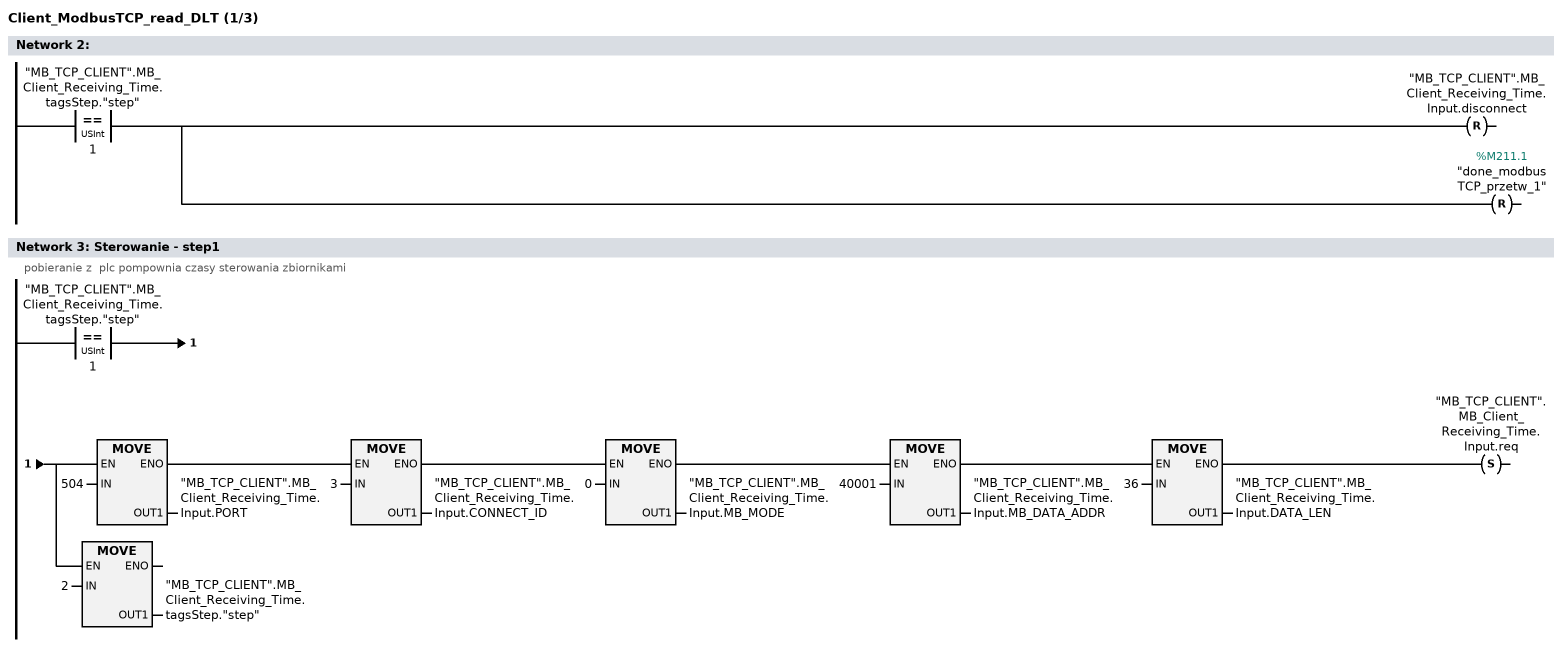
   RUNG wire#powerrail
      { S7_Templates := "SrcType := USInt" } EQ_Contact(in1 := "MB_TCP_CLIENT".MB_Client_Receiving_Time.tagsStep."step", in2 := 1)
      wire#w1
      R_Coil( "MB_TCP_CLIENT".MB_Client_Receiving_Time.Input.disconnect )
   END_RUNG
   RUNG wire#w1
      R_Coil( "done_modbusTCP_przetw_1" )
   END_RUNG
   // the same network as SCL:
   IF "MB_TCP_CLIENT".MB_Client_Receiving_Time.tagsStep."step" = 1 THEN
       "MB_TCP_CLIENT".MB_Client_Receiving_Time.Input.disconnect := FALSE;
       "done_modbusTCP_przetw_1" := FALSE;
   END_IF;
END_REGION

REGION Network 3: Sterowanie - step1
   // pobieranie z  plc pompownia czasy sterowania zbiornikami
   RUNG wire#powerrail
      { S7_Templates := "SrcType := USInt" } EQ_Contact(in1 := "MB_TCP_CLIENT".MB_Client_Receiving_Time.tagsStep."step", in2 := 1)
      wire#w1
      { S7_GenerateENO := "TRUE" } Move(in := 504, out1 => "MB_TCP_CLIENT".MB_Client_Receiving_Time.Input.PORT)
      { S7_GenerateENO := "TRUE" } Move(in := 3, out1 => "MB_TCP_CLIENT".MB_Client_Receiving_Time.Input.CONNECT_ID)
      { S7_GenerateENO := "TRUE" } Move(in := 0, out1 => "MB_TCP_CLIENT".MB_Client_Receiving_Time.Input.MB_MODE)
      { S7_GenerateENO := "TRUE" } Move(in := 40001, out1 => "MB_TCP_CLIENT".MB_Client_Receiving_Time.Input.MB_DATA_ADDR)
      { S7_GenerateENO := "TRUE" } Move(in := 36, out1 => "MB_TCP_CLIENT".MB_Client_Receiving_Time.Input.DATA_LEN)
      S_Coil( "MB_TCP_CLIENT".MB_Client_Receiving_Time.Input.req )
   END_RUNG
   RUNG wire#w1
      { S7_GenerateENO := "TRUE" } Move(in := 2, out1 => "MB_TCP_CLIENT".MB_Client_Receiving_Time.tagsStep."step")
   END_RUNG
   // the same network as SCL:
   // ENO of a box is taken as its EN; it also drops when the box reports an error
   IF "MB_TCP_CLIENT".MB_Client_Receiving_Time.tagsStep."step" = 1 THEN
       "MB_TCP_CLIENT".MB_Client_Receiving_Time.Input.PORT := 504;
       "MB_TCP_CLIENT".MB_Client_Receiving_Time.Input.CONNECT_ID := 3;
       "MB_TCP_CLIENT".MB_Client_Receiving_Time.Input.MB_MODE := 0;
       "MB_TCP_CLIENT".MB_Client_Receiving_Time.Input.MB_DATA_ADDR := 40001;
       "MB_TCP_CLIENT".MB_Client_Receiving_Time.Input.DATA_LEN := 36;
       "MB_TCP_CLIENT".MB_Client_Receiving_Time.Input.req := TRUE;
       "MB_TCP_CLIENT".MB_Client_Receiving_Time.tagsStep."step" := 2;
   END_IF;
END_REGION

REGION Network 4: step 2
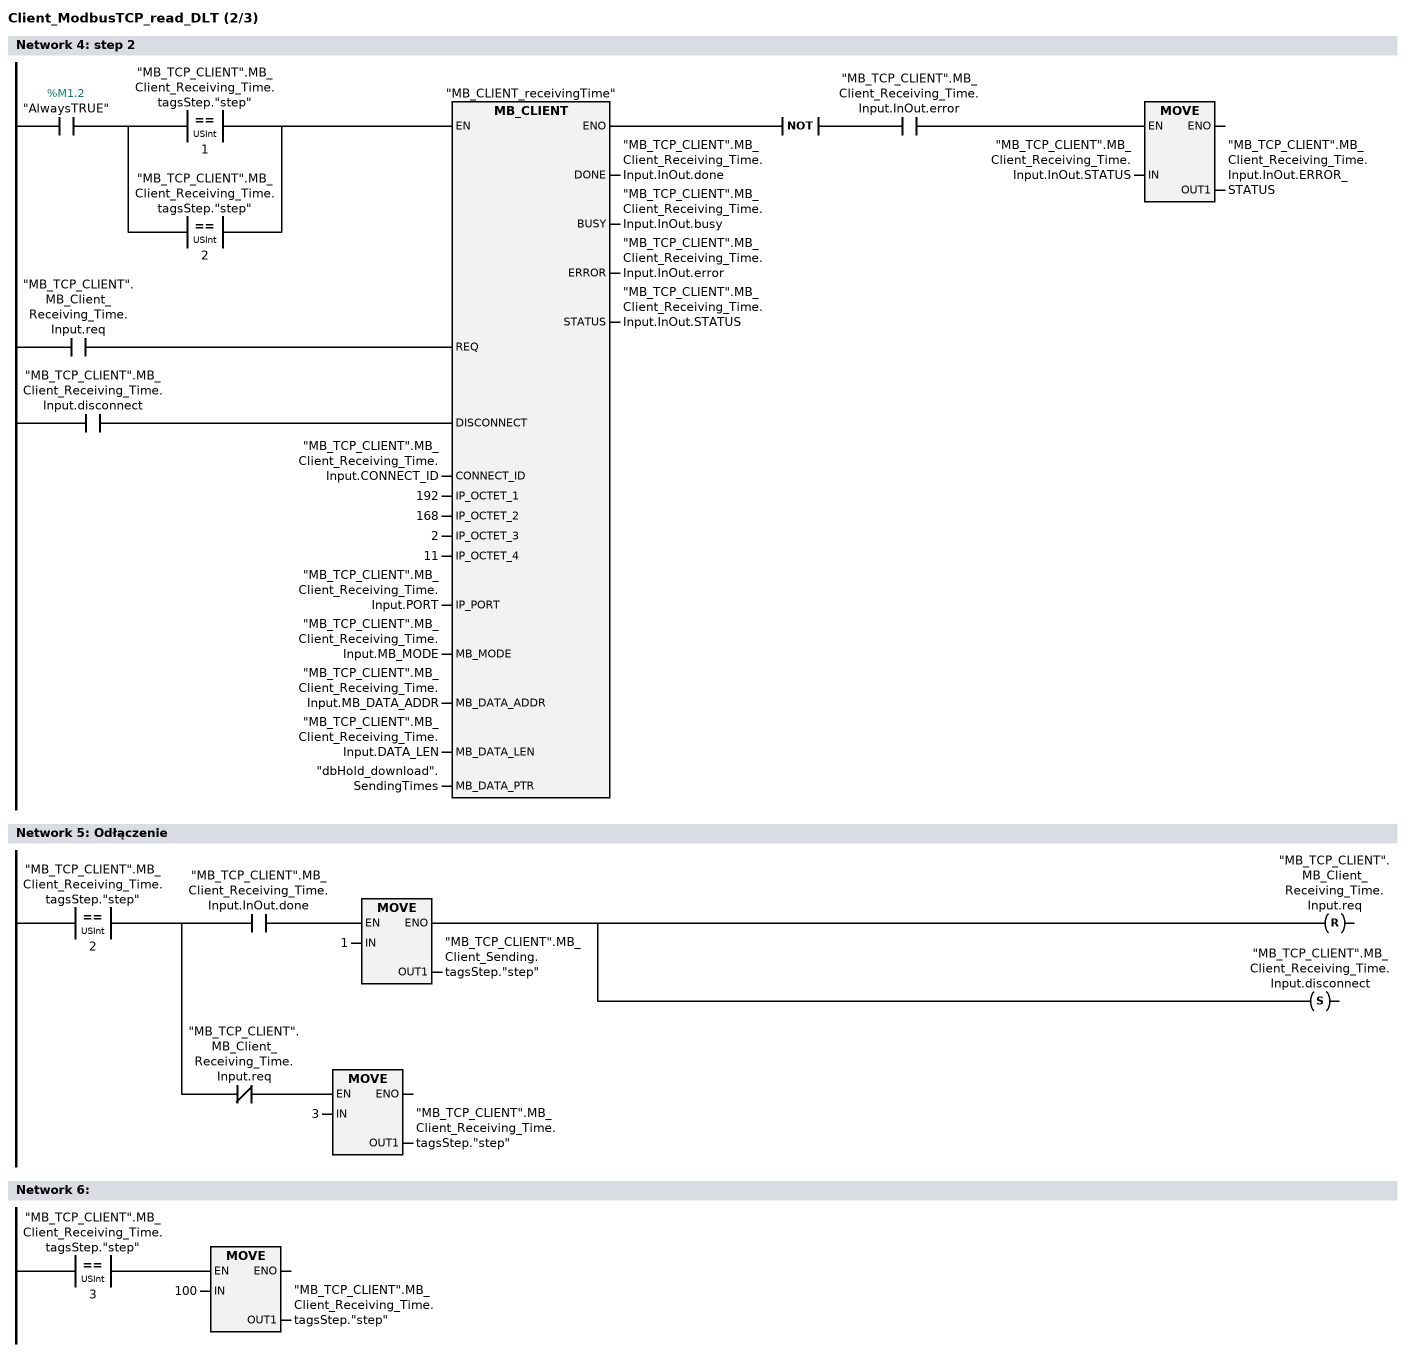
   RUNG wire#powerrail
      Contact( "AlwaysTRUE" )
      wire#w1
      { S7_Templates := "SrcType := USInt" } EQ_Contact(in1 := "MB_TCP_CLIENT".MB_Client_Receiving_Time.tagsStep."step", in2 := 1)
      wire#w2
      { S7_Templates := "[card1200 := 1, card1500 := 0]" } "MB_CLIENT_receivingTime".MB_CLIENT(REQ := wire#w3, DISCONNECT := wire#w4, CONNECT_ID := "MB_TCP_CLIENT".MB_Client_Receiving_Time.Input.CONNECT_ID, IP_OCTET_1 := 192, IP_OCTET_2 := 168, IP_OCTET_3 := 2, IP_OCTET_4 := 11, IP_PORT := "MB_TCP_CLIENT".MB_Client_Receiving_Time.Input.PORT, MB_MODE := "MB_TCP_CLIENT".MB_Client_Receiving_Time.Input.MB_MODE, MB_DATA_ADDR := "MB_TCP_CLIENT".MB_Client_Receiving_Time.Input.MB_DATA_ADDR, MB_DATA_LEN := "MB_TCP_CLIENT".MB_Client_Receiving_Time.Input.DATA_LEN, MB_DATA_PTR := "dbHold_download".SendingTimes, DONE => "MB_TCP_CLIENT".MB_Client_Receiving_Time.Input.InOut.done, BUSY => "MB_TCP_CLIENT".MB_Client_Receiving_Time.Input.InOut.busy, ERROR => "MB_TCP_CLIENT".MB_Client_Receiving_Time.Input.InOut.error, STATUS => "MB_TCP_CLIENT".MB_Client_Receiving_Time.Input.InOut.STATUS)
      Not()
      Contact( "MB_TCP_CLIENT".MB_Client_Receiving_Time.Input.InOut.error )
      Move(in := "MB_TCP_CLIENT".MB_Client_Receiving_Time.Input.InOut.STATUS, out1 => "MB_TCP_CLIENT".MB_Client_Receiving_Time.Input.InOut.ERROR_STATUS)
   END_RUNG
   RUNG wire#w1
      { S7_Templates := "SrcType := USInt" } EQ_Contact(in1 := "MB_TCP_CLIENT".MB_Client_Receiving_Time.tagsStep."step", in2 := 2)
   END_RUNG wire#w2
   RUNG wire#powerrail
      Contact( "MB_TCP_CLIENT".MB_Client_Receiving_Time.Input.req )
   END_RUNG wire#w3
   RUNG wire#powerrail
      Contact( "MB_TCP_CLIENT".MB_Client_Receiving_Time.Input.disconnect )
   END_RUNG wire#w4
   // the same network as SCL:
   #_w1 := "AlwaysTRUE" AND (("MB_TCP_CLIENT".MB_Client_Receiving_Time.tagsStep."step" = 1) OR ("MB_TCP_CLIENT".MB_Client_Receiving_Time.tagsStep."step" = 2));
   "MB_CLIENT_receivingTime"(EN := #_w1,   // MB_CLIENT
                           REQ := "MB_TCP_CLIENT".MB_Client_Receiving_Time.Input.req,
                           DISCONNECT := "MB_TCP_CLIENT".MB_Client_Receiving_Time.Input.disconnect,
                           CONNECT_ID := "MB_TCP_CLIENT".MB_Client_Receiving_Time.Input.CONNECT_ID,
                           IP_OCTET_1 := 192,
                           IP_OCTET_2 := 168,
                           IP_OCTET_3 := 2,
                           IP_OCTET_4 := 11,
                           IP_PORT := "MB_TCP_CLIENT".MB_Client_Receiving_Time.Input.PORT,
                           MB_MODE := "MB_TCP_CLIENT".MB_Client_Receiving_Time.Input.MB_MODE,
                           MB_DATA_ADDR := "MB_TCP_CLIENT".MB_Client_Receiving_Time.Input.MB_DATA_ADDR,
                           MB_DATA_LEN := "MB_TCP_CLIENT".MB_Client_Receiving_Time.Input.DATA_LEN,
                           MB_DATA_PTR := "dbHold_download".SendingTimes,
                           DONE => "MB_TCP_CLIENT".MB_Client_Receiving_Time.Input.InOut.done,
                           BUSY => "MB_TCP_CLIENT".MB_Client_Receiving_Time.Input.InOut.busy,
                           ERROR => "MB_TCP_CLIENT".MB_Client_Receiving_Time.Input.InOut.error,
                           STATUS => "MB_TCP_CLIENT".MB_Client_Receiving_Time.Input.InOut.STATUS,
                           ENO => #_w2);
   IF NOT #_w2 AND "MB_TCP_CLIENT".MB_Client_Receiving_Time.Input.InOut.error THEN
       "MB_TCP_CLIENT".MB_Client_Receiving_Time.Input.InOut.ERROR_STATUS := "MB_TCP_CLIENT".MB_Client_Receiving_Time.Input.InOut.STATUS;
   END_IF;
END_REGION

REGION Network 5: Odłączenie
   RUNG wire#powerrail
      { S7_Templates := "SrcType := USInt" } EQ_Contact(in1 := "MB_TCP_CLIENT".MB_Client_Receiving_Time.tagsStep."step", in2 := 2)
      wire#w1
      Contact( "MB_TCP_CLIENT".MB_Client_Receiving_Time.Input.InOut.done )
      Move(in := 1, out1 => "MB_TCP_CLIENT".MB_Client_Sending.tagsStep."step")
      wire#w2
      R_Coil( "MB_TCP_CLIENT".MB_Client_Receiving_Time.Input.req )
   END_RUNG
   RUNG wire#w2
      S_Coil( "MB_TCP_CLIENT".MB_Client_Receiving_Time.Input.disconnect )
   END_RUNG
   RUNG wire#w1
      I_Contact( "MB_TCP_CLIENT".MB_Client_Receiving_Time.Input.req )
      Move(in := 3, out1 => "MB_TCP_CLIENT".MB_Client_Receiving_Time.tagsStep."step")
   END_RUNG
   // the same network as SCL:
   #_w1 := "MB_TCP_CLIENT".MB_Client_Receiving_Time.tagsStep."step" = 2;
   IF #_w1 AND "MB_TCP_CLIENT".MB_Client_Receiving_Time.Input.InOut.done THEN
       "MB_TCP_CLIENT".MB_Client_Sending.tagsStep."step" := 1;
       "MB_TCP_CLIENT".MB_Client_Receiving_Time.Input.req := FALSE;
       "MB_TCP_CLIENT".MB_Client_Receiving_Time.Input.disconnect := TRUE;
   END_IF;
   IF #_w1 AND NOT "MB_TCP_CLIENT".MB_Client_Receiving_Time.Input.req THEN
       "MB_TCP_CLIENT".MB_Client_Receiving_Time.tagsStep."step" := 3;
   END_IF;
END_REGION

REGION Network 6
   RUNG wire#powerrail
      { S7_Templates := "SrcType := USInt" } EQ_Contact(in1 := "MB_TCP_CLIENT".MB_Client_Receiving_Time.tagsStep."step", in2 := 3)
      Move(in := 100, out1 => "MB_TCP_CLIENT".MB_Client_Receiving_Time.tagsStep."step")
   END_RUNG
   // the same network as SCL:
   IF "MB_TCP_CLIENT".MB_Client_Receiving_Time.tagsStep."step" = 3 THEN
       "MB_TCP_CLIENT".MB_Client_Receiving_Time.tagsStep."step" := 100;
   END_IF;
END_REGION

REGION Network 7
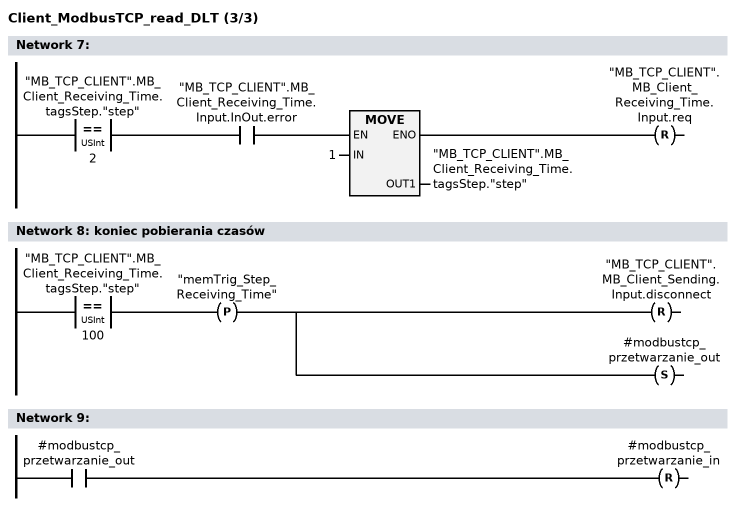
   RUNG wire#powerrail
      { S7_Templates := "SrcType := USInt" } EQ_Contact(in1 := "MB_TCP_CLIENT".MB_Client_Receiving_Time.tagsStep."step", in2 := 2)
      Contact( "MB_TCP_CLIENT".MB_Client_Receiving_Time.Input.InOut.error )
      Move(in := 1, out1 => "MB_TCP_CLIENT".MB_Client_Receiving_Time.tagsStep."step")
      R_Coil( "MB_TCP_CLIENT".MB_Client_Receiving_Time.Input.req )
   END_RUNG
   // the same network as SCL:
   #_w1 := ("MB_TCP_CLIENT".MB_Client_Receiving_Time.tagsStep."step" = 2) AND "MB_TCP_CLIENT".MB_Client_Receiving_Time.Input.InOut.error;
   IF #_w1 THEN
       "MB_TCP_CLIENT".MB_Client_Receiving_Time.tagsStep."step" := 1;
       "MB_TCP_CLIENT".MB_Client_Receiving_Time.Input.req := FALSE;
   END_IF;
END_REGION

REGION Network 8: koniec pobierania czasów
   RUNG wire#powerrail
      { S7_Templates := "SrcType := USInt" } EQ_Contact(in1 := "MB_TCP_CLIENT".MB_Client_Receiving_Time.tagsStep."step", in2 := 100)
      P_Trig( "memTrig_Step_Receiving_Time" )
      wire#w1
      R_Coil( "MB_TCP_CLIENT".MB_Client_Sending.Input.disconnect )
   END_RUNG
   RUNG wire#w1
      S_Coil( #modbustcp_przetwarzanie_out )
   END_RUNG
   // the same network as SCL:
   #_w1 := "MB_TCP_CLIENT".MB_Client_Receiving_Time.tagsStep."step" = 100;
   #_w2 := #_w1 AND NOT "memTrig_Step_Receiving_Time";   // rising edge
   "memTrig_Step_Receiving_Time" := #_w1;
   IF #_w2 THEN
       "MB_TCP_CLIENT".MB_Client_Sending.Input.disconnect := FALSE;
       #modbustcp_przetwarzanie_out := TRUE;
   END_IF;
END_REGION

REGION Network 9
   RUNG wire#powerrail
      Contact( #modbustcp_przetwarzanie_out )
      R_Coil( #modbustcp_przetwarzanie_in )
   END_RUNG
   // the same network as SCL:
   IF #modbustcp_przetwarzanie_out THEN #modbustcp_przetwarzanie_in := FALSE; END_IF;
END_REGION
END_FUNCTION_BLOCK

FUNCTION_BLOCK "Client_ModbusTCP_sending_analogs"   // FB4, LAD
TITLE = Wysyłanie analogów
{ S7_Optimized_Access := 'TRUE' }
AUTHOR : rtecmer
VERSION : 0.1
// Wysyłanie pomiarów
// stored: AutoNumber true, IsIECCheckEnabled false, IsRetainMemResEnabled false, MemoryReserve 250, SetENOAutomatically false, UDAEnableTagReadback false
   VAR_IN_OUT
      modbustcp_przetwarzanie_in : Bool;
      modbustcp_przetwarzanie_out : Bool;
   END_VAR
   VAR_TEMP   // added for the SCL form of the ladder/FBD networks
      _w1 : Bool;
      _w2 : Bool;
   END_VAR
BEGIN

REGION Network 2: Inicjacja modbus po błędzie i restarcie
END_REGION

REGION Network 3
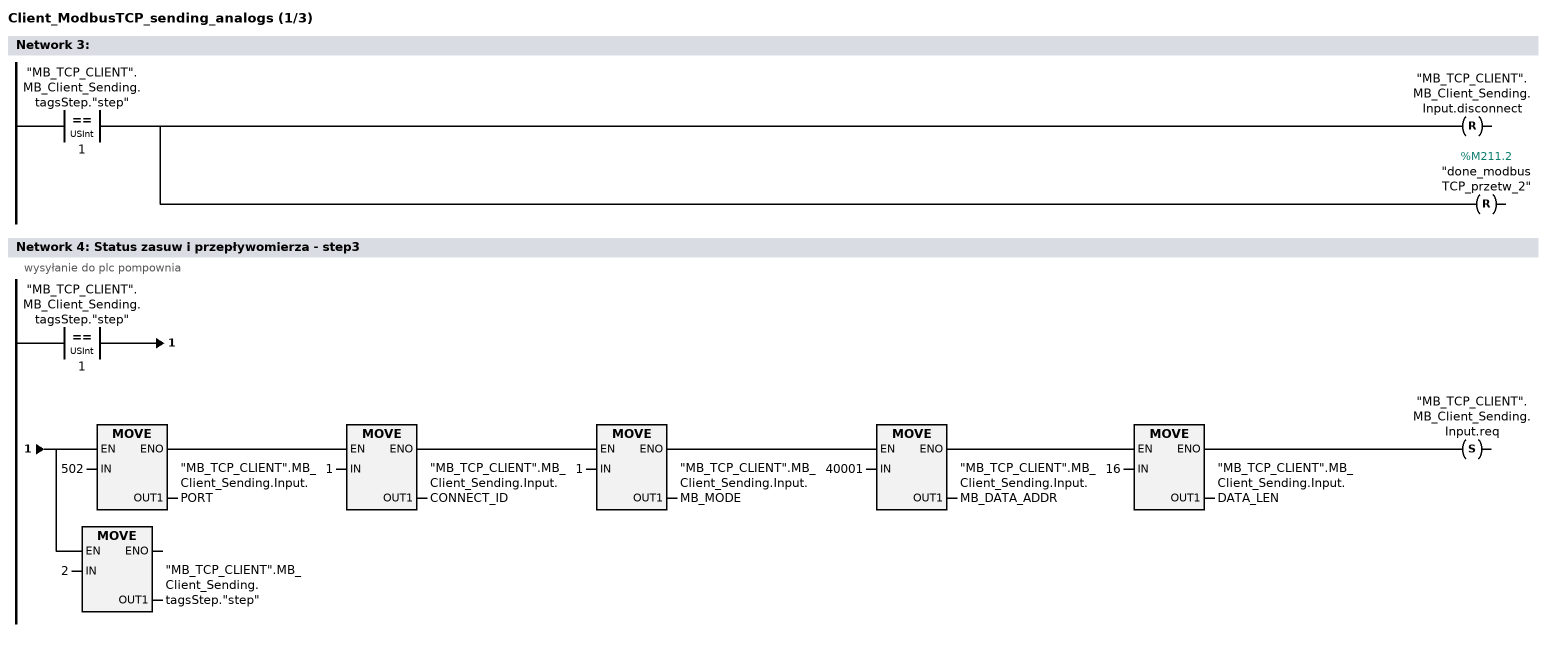
   RUNG wire#powerrail
      { S7_Templates := "SrcType := USInt" } EQ_Contact(in1 := "MB_TCP_CLIENT".MB_Client_Sending.tagsStep."step", in2 := 1)
      wire#w1
      R_Coil( "MB_TCP_CLIENT".MB_Client_Sending.Input.disconnect )
   END_RUNG
   RUNG wire#w1
      R_Coil( "done_modbusTCP_przetw_2" )
   END_RUNG
   // the same network as SCL:
   IF "MB_TCP_CLIENT".MB_Client_Sending.tagsStep."step" = 1 THEN
       "MB_TCP_CLIENT".MB_Client_Sending.Input.disconnect := FALSE;
       "done_modbusTCP_przetw_2" := FALSE;
   END_IF;
END_REGION

REGION Network 4: Status zasuw i przepływomierza - step3
   // wysyłanie do plc pompownia
   RUNG wire#powerrail
      { S7_Templates := "SrcType := USInt" } EQ_Contact(in1 := "MB_TCP_CLIENT".MB_Client_Sending.tagsStep."step", in2 := 1)
      wire#w1
      { S7_GenerateENO := "TRUE" } Move(in := 502, out1 => "MB_TCP_CLIENT".MB_Client_Sending.Input.PORT)
      { S7_GenerateENO := "TRUE" } Move(in := 1, out1 => "MB_TCP_CLIENT".MB_Client_Sending.Input.CONNECT_ID)
      { S7_GenerateENO := "TRUE" } Move(in := 1, out1 => "MB_TCP_CLIENT".MB_Client_Sending.Input.MB_MODE)
      { S7_GenerateENO := "TRUE" } Move(in := 40001, out1 => "MB_TCP_CLIENT".MB_Client_Sending.Input.MB_DATA_ADDR)
      { S7_GenerateENO := "TRUE" } Move(in := 16, out1 => "MB_TCP_CLIENT".MB_Client_Sending.Input.DATA_LEN)
      S_Coil( "MB_TCP_CLIENT".MB_Client_Sending.Input.req )
   END_RUNG
   RUNG wire#w1
      { S7_GenerateENO := "TRUE" } Move(in := 2, out1 => "MB_TCP_CLIENT".MB_Client_Sending.tagsStep."step")
   END_RUNG
   // the same network as SCL:
   // ENO of a box is taken as its EN; it also drops when the box reports an error
   IF "MB_TCP_CLIENT".MB_Client_Sending.tagsStep."step" = 1 THEN
       "MB_TCP_CLIENT".MB_Client_Sending.Input.PORT := 502;
       "MB_TCP_CLIENT".MB_Client_Sending.Input.CONNECT_ID := 1;
       "MB_TCP_CLIENT".MB_Client_Sending.Input.MB_MODE := 1;
       "MB_TCP_CLIENT".MB_Client_Sending.Input.MB_DATA_ADDR := 40001;
       "MB_TCP_CLIENT".MB_Client_Sending.Input.DATA_LEN := 16;
       "MB_TCP_CLIENT".MB_Client_Sending.Input.req := TRUE;
       "MB_TCP_CLIENT".MB_Client_Sending.tagsStep."step" := 2;
   END_IF;
END_REGION

REGION Network 5: step 3
   // Analogi
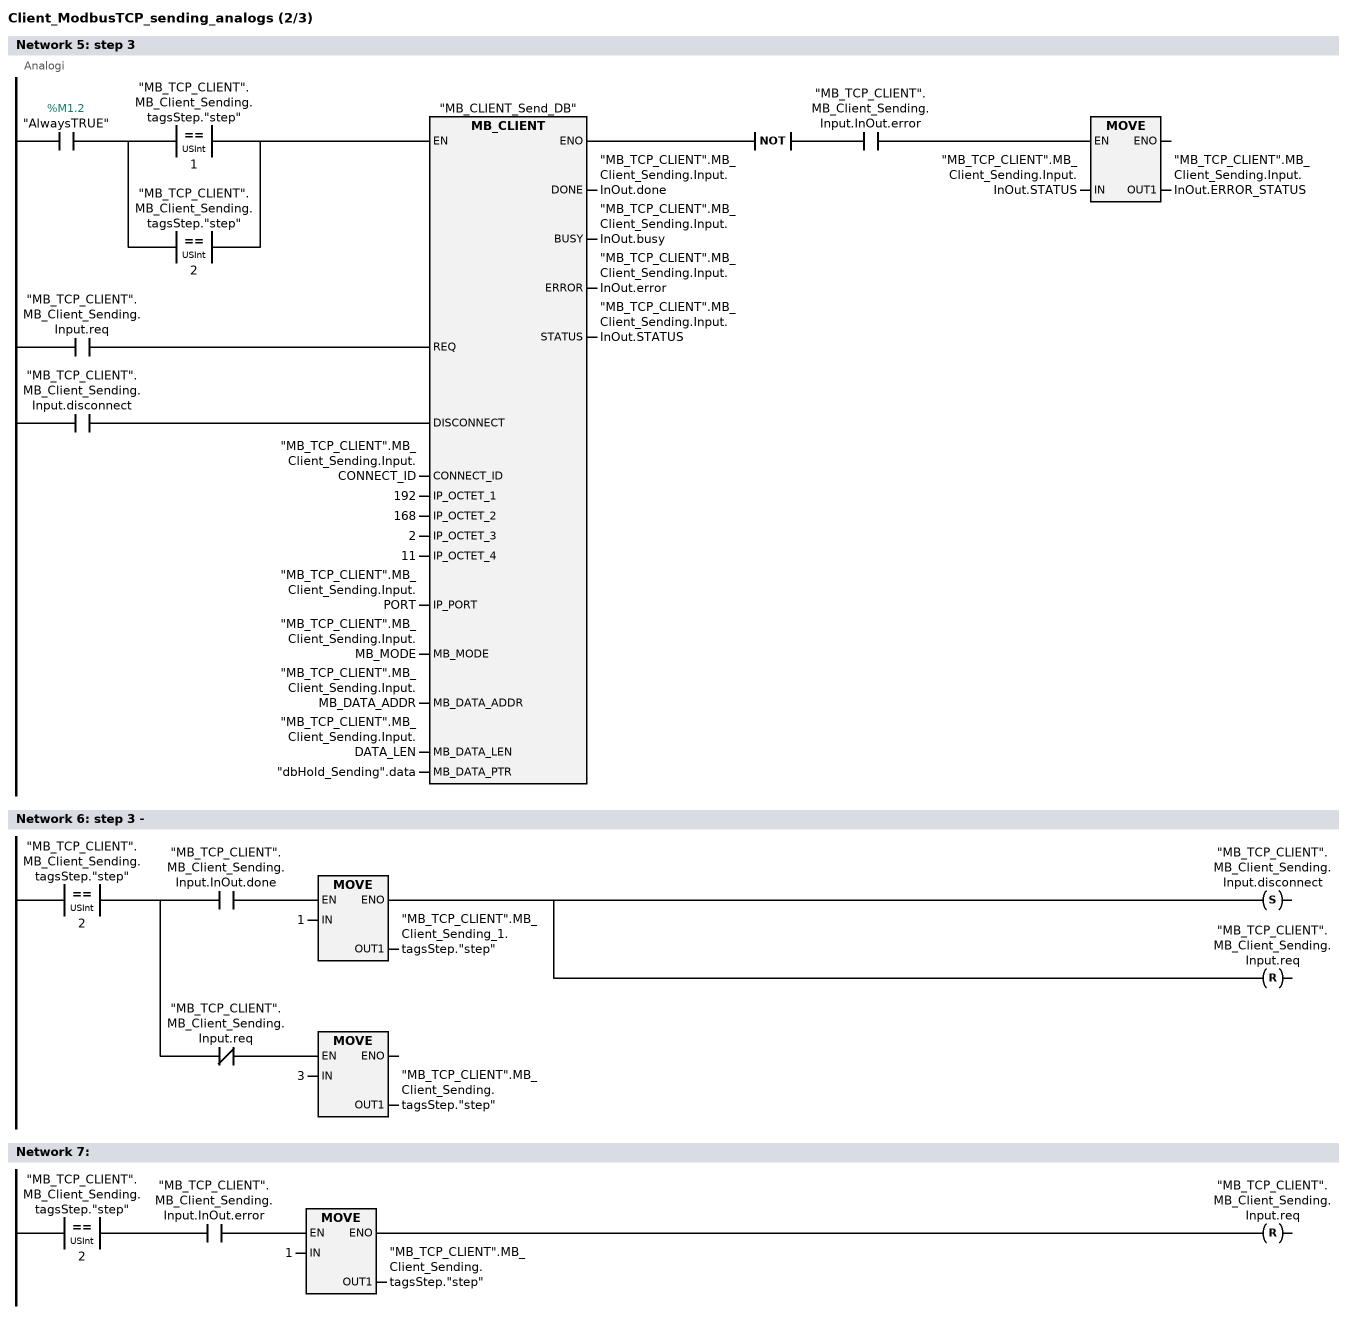
   RUNG wire#powerrail
      Contact( "AlwaysTRUE" )
      wire#w1
      { S7_Templates := "SrcType := USInt" } EQ_Contact(in1 := "MB_TCP_CLIENT".MB_Client_Sending.tagsStep."step", in2 := 1)
      wire#w2
      { S7_Templates := "[card1200 := 1, card1500 := 0]" } "MB_CLIENT_Send_DB".MB_CLIENT(REQ := wire#w3, DISCONNECT := wire#w4, CONNECT_ID := "MB_TCP_CLIENT".MB_Client_Sending.Input.CONNECT_ID, IP_OCTET_1 := 192, IP_OCTET_2 := 168, IP_OCTET_3 := 2, IP_OCTET_4 := 11, IP_PORT := "MB_TCP_CLIENT".MB_Client_Sending.Input.PORT, MB_MODE := "MB_TCP_CLIENT".MB_Client_Sending.Input.MB_MODE, MB_DATA_ADDR := "MB_TCP_CLIENT".MB_Client_Sending.Input.MB_DATA_ADDR, MB_DATA_LEN := "MB_TCP_CLIENT".MB_Client_Sending.Input.DATA_LEN, MB_DATA_PTR := "dbHold_Sending".data, DONE => "MB_TCP_CLIENT".MB_Client_Sending.Input.InOut.done, BUSY => "MB_TCP_CLIENT".MB_Client_Sending.Input.InOut.busy, ERROR => "MB_TCP_CLIENT".MB_Client_Sending.Input.InOut.error, STATUS => "MB_TCP_CLIENT".MB_Client_Sending.Input.InOut.STATUS)
      Not()
      Contact( "MB_TCP_CLIENT".MB_Client_Sending.Input.InOut.error )
      Move(in := "MB_TCP_CLIENT".MB_Client_Sending.Input.InOut.STATUS, out1 => "MB_TCP_CLIENT".MB_Client_Sending.Input.InOut.ERROR_STATUS)
   END_RUNG
   RUNG wire#w1
      { S7_Templates := "SrcType := USInt" } EQ_Contact(in1 := "MB_TCP_CLIENT".MB_Client_Sending.tagsStep."step", in2 := 2)
   END_RUNG wire#w2
   RUNG wire#powerrail
      Contact( "MB_TCP_CLIENT".MB_Client_Sending.Input.req )
   END_RUNG wire#w3
   RUNG wire#powerrail
      Contact( "MB_TCP_CLIENT".MB_Client_Sending.Input.disconnect )
   END_RUNG wire#w4
   // the same network as SCL:
   #_w1 := "AlwaysTRUE" AND (("MB_TCP_CLIENT".MB_Client_Sending.tagsStep."step" = 1) OR ("MB_TCP_CLIENT".MB_Client_Sending.tagsStep."step" = 2));
   "MB_CLIENT_Send_DB"(EN := #_w1,   // MB_CLIENT
                       REQ := "MB_TCP_CLIENT".MB_Client_Sending.Input.req,
                       DISCONNECT := "MB_TCP_CLIENT".MB_Client_Sending.Input.disconnect,
                       CONNECT_ID := "MB_TCP_CLIENT".MB_Client_Sending.Input.CONNECT_ID,
                       IP_OCTET_1 := 192,
                       IP_OCTET_2 := 168,
                       IP_OCTET_3 := 2,
                       IP_OCTET_4 := 11,
                       IP_PORT := "MB_TCP_CLIENT".MB_Client_Sending.Input.PORT,
                       MB_MODE := "MB_TCP_CLIENT".MB_Client_Sending.Input.MB_MODE,
                       MB_DATA_ADDR := "MB_TCP_CLIENT".MB_Client_Sending.Input.MB_DATA_ADDR,
                       MB_DATA_LEN := "MB_TCP_CLIENT".MB_Client_Sending.Input.DATA_LEN,
                       MB_DATA_PTR := "dbHold_Sending".data,
                       DONE => "MB_TCP_CLIENT".MB_Client_Sending.Input.InOut.done,
                       BUSY => "MB_TCP_CLIENT".MB_Client_Sending.Input.InOut.busy,
                       ERROR => "MB_TCP_CLIENT".MB_Client_Sending.Input.InOut.error,
                       STATUS => "MB_TCP_CLIENT".MB_Client_Sending.Input.InOut.STATUS,
                       ENO => #_w2);
   IF NOT #_w2 AND "MB_TCP_CLIENT".MB_Client_Sending.Input.InOut.error THEN
       "MB_TCP_CLIENT".MB_Client_Sending.Input.InOut.ERROR_STATUS := "MB_TCP_CLIENT".MB_Client_Sending.Input.InOut.STATUS;
   END_IF;
END_REGION

REGION Network 6: step 3 -
   RUNG wire#powerrail
      { S7_Templates := "SrcType := USInt" } EQ_Contact(in1 := "MB_TCP_CLIENT".MB_Client_Sending.tagsStep."step", in2 := 2)
      wire#w1
      Contact( "MB_TCP_CLIENT".MB_Client_Sending.Input.InOut.done )
      Move(in := 1, out1 => "MB_TCP_CLIENT".MB_Client_Sending_1.tagsStep."step")
      wire#w2
      S_Coil( "MB_TCP_CLIENT".MB_Client_Sending.Input.disconnect )
   END_RUNG
   RUNG wire#w2
      R_Coil( "MB_TCP_CLIENT".MB_Client_Sending.Input.req )
   END_RUNG
   RUNG wire#w1
      I_Contact( "MB_TCP_CLIENT".MB_Client_Sending.Input.req )
      Move(in := 3, out1 => "MB_TCP_CLIENT".MB_Client_Sending.tagsStep."step")
   END_RUNG
   // the same network as SCL:
   #_w1 := "MB_TCP_CLIENT".MB_Client_Sending.tagsStep."step" = 2;
   IF #_w1 AND "MB_TCP_CLIENT".MB_Client_Sending.Input.InOut.done THEN
       "MB_TCP_CLIENT".MB_Client_Sending_1.tagsStep."step" := 1;
       "MB_TCP_CLIENT".MB_Client_Sending.Input.disconnect := TRUE;
       "MB_TCP_CLIENT".MB_Client_Sending.Input.req := FALSE;
   END_IF;
   IF #_w1 AND NOT "MB_TCP_CLIENT".MB_Client_Sending.Input.req THEN
       "MB_TCP_CLIENT".MB_Client_Sending.tagsStep."step" := 3;
   END_IF;
END_REGION

REGION Network 7
   RUNG wire#powerrail
      { S7_Templates := "SrcType := USInt" } EQ_Contact(in1 := "MB_TCP_CLIENT".MB_Client_Sending.tagsStep."step", in2 := 2)
      Contact( "MB_TCP_CLIENT".MB_Client_Sending.Input.InOut.error )
      Move(in := 1, out1 => "MB_TCP_CLIENT".MB_Client_Sending.tagsStep."step")
      R_Coil( "MB_TCP_CLIENT".MB_Client_Sending.Input.req )
   END_RUNG
   // the same network as SCL:
   #_w1 := ("MB_TCP_CLIENT".MB_Client_Sending.tagsStep."step" = 2) AND "MB_TCP_CLIENT".MB_Client_Sending.Input.InOut.error;
   IF #_w1 THEN
       "MB_TCP_CLIENT".MB_Client_Sending.tagsStep."step" := 1;
       "MB_TCP_CLIENT".MB_Client_Sending.Input.req := FALSE;
   END_IF;
END_REGION

REGION Network 8
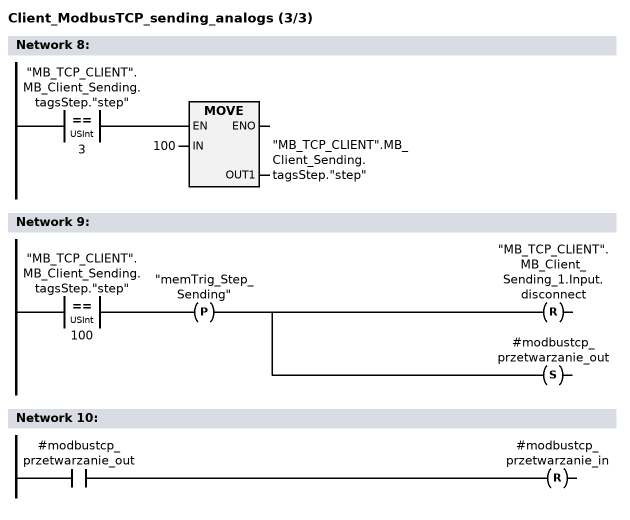
   RUNG wire#powerrail
      { S7_Templates := "SrcType := USInt" } EQ_Contact(in1 := "MB_TCP_CLIENT".MB_Client_Sending.tagsStep."step", in2 := 3)
      Move(in := 100, out1 => "MB_TCP_CLIENT".MB_Client_Sending.tagsStep."step")
   END_RUNG
   // the same network as SCL:
   IF "MB_TCP_CLIENT".MB_Client_Sending.tagsStep."step" = 3 THEN
       "MB_TCP_CLIENT".MB_Client_Sending.tagsStep."step" := 100;
   END_IF;
END_REGION

REGION Network 9
   RUNG wire#powerrail
      { S7_Templates := "SrcType := USInt" } EQ_Contact(in1 := "MB_TCP_CLIENT".MB_Client_Sending.tagsStep."step", in2 := 100)
      P_Trig( "memTrig_Step_Sending" )
      wire#w1
      R_Coil( "MB_TCP_CLIENT".MB_Client_Sending_1.Input.disconnect )
   END_RUNG
   RUNG wire#w1
      S_Coil( #modbustcp_przetwarzanie_out )
   END_RUNG
   // the same network as SCL:
   #_w1 := "MB_TCP_CLIENT".MB_Client_Sending.tagsStep."step" = 100;
   #_w2 := #_w1 AND NOT "memTrig_Step_Sending";   // rising edge
   "memTrig_Step_Sending" := #_w1;
   IF #_w2 THEN
       "MB_TCP_CLIENT".MB_Client_Sending_1.Input.disconnect := FALSE;
       #modbustcp_przetwarzanie_out := TRUE;
   END_IF;
END_REGION

REGION Network 10
   RUNG wire#powerrail
      Contact( #modbustcp_przetwarzanie_out )
      R_Coil( #modbustcp_przetwarzanie_in )
   END_RUNG
   // the same network as SCL:
   IF #modbustcp_przetwarzanie_out THEN #modbustcp_przetwarzanie_in := FALSE; END_IF;
END_REGION
END_FUNCTION_BLOCK

FUNCTION_BLOCK "Client_ModbusTCP_sending_status"   // FB8, LAD
TITLE = Przekazanie statusu utrządzeń
{ S7_Optimized_Access := 'TRUE' }
AUTHOR : rtecmer
VERSION : 0.1
// funkcja przesyła na server status urządzeńz PLC 2 Zbiorniki
// stored: AutoNumber true, IsIECCheckEnabled false, IsRetainMemResEnabled false, MemoryReserve 250, SetENOAutomatically false, UDAEnableTagReadback false
   VAR_IN_OUT
      modbustcp_przetwarzanie_in : Bool;
      modbustcp_przetwarzanie_out : Bool;
   END_VAR
   VAR_TEMP   // added for the SCL form of the ladder/FBD networks
      _w1 : Bool;
      _w2 : Bool;
   END_VAR
BEGIN

REGION Network 1: Inicjacja modbus po błędzie i restarcie
END_REGION

REGION Network 2
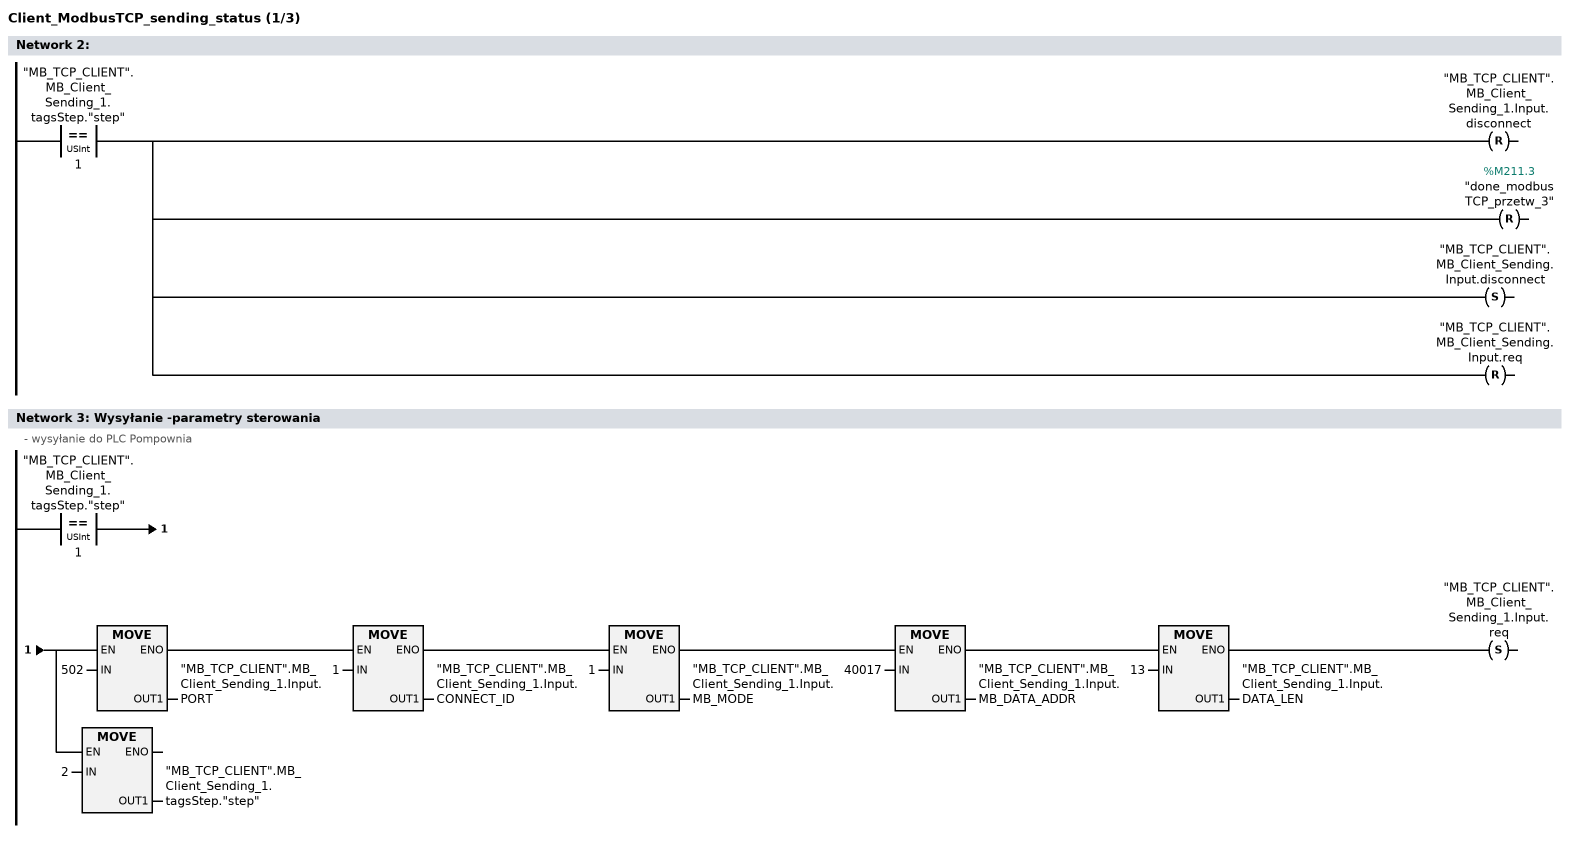
   RUNG wire#powerrail
      { S7_Templates := "SrcType := USInt" } EQ_Contact(in1 := "MB_TCP_CLIENT".MB_Client_Sending_1.tagsStep."step", in2 := 1)
      wire#w1
      R_Coil( "MB_TCP_CLIENT".MB_Client_Sending_1.Input.disconnect )
   END_RUNG
   RUNG wire#w1
      R_Coil( "done_modbusTCP_przetw_3" )
   END_RUNG
   RUNG wire#w1
      S_Coil( "MB_TCP_CLIENT".MB_Client_Sending.Input.disconnect )
   END_RUNG
   RUNG wire#w1
      R_Coil( "MB_TCP_CLIENT".MB_Client_Sending.Input.req )
   END_RUNG
   // the same network as SCL:
   IF "MB_TCP_CLIENT".MB_Client_Sending_1.tagsStep."step" = 1 THEN
       "MB_TCP_CLIENT".MB_Client_Sending_1.Input.disconnect := FALSE;
       "done_modbusTCP_przetw_3" := FALSE;
       "MB_TCP_CLIENT".MB_Client_Sending.Input.disconnect := TRUE;
       "MB_TCP_CLIENT".MB_Client_Sending.Input.req := FALSE;
   END_IF;
END_REGION

REGION Network 3: Wysyłanie -parametry sterowania
   // - wysyłanie do PLC Pompownia
   RUNG wire#powerrail
      { S7_Templates := "SrcType := USInt" } EQ_Contact(in1 := "MB_TCP_CLIENT".MB_Client_Sending_1.tagsStep."step", in2 := 1)
      wire#w1
      { S7_GenerateENO := "TRUE" } Move(in := 502, out1 => "MB_TCP_CLIENT".MB_Client_Sending_1.Input.PORT)
      { S7_GenerateENO := "TRUE" } Move(in := 1, out1 => "MB_TCP_CLIENT".MB_Client_Sending_1.Input.CONNECT_ID)
      { S7_GenerateENO := "TRUE" } Move(in := 1, out1 => "MB_TCP_CLIENT".MB_Client_Sending_1.Input.MB_MODE)
      { S7_GenerateENO := "TRUE" } Move(in := 40017, out1 => "MB_TCP_CLIENT".MB_Client_Sending_1.Input.MB_DATA_ADDR)
      { S7_GenerateENO := "TRUE" } Move(in := 13, out1 => "MB_TCP_CLIENT".MB_Client_Sending_1.Input.DATA_LEN)
      S_Coil( "MB_TCP_CLIENT".MB_Client_Sending_1.Input.req )
   END_RUNG
   RUNG wire#w1
      { S7_GenerateENO := "TRUE" } Move(in := 2, out1 => "MB_TCP_CLIENT".MB_Client_Sending_1.tagsStep."step")
   END_RUNG
   // the same network as SCL:
   // ENO of a box is taken as its EN; it also drops when the box reports an error
   IF "MB_TCP_CLIENT".MB_Client_Sending_1.tagsStep."step" = 1 THEN
       "MB_TCP_CLIENT".MB_Client_Sending_1.Input.PORT := 502;
       "MB_TCP_CLIENT".MB_Client_Sending_1.Input.CONNECT_ID := 1;
       "MB_TCP_CLIENT".MB_Client_Sending_1.Input.MB_MODE := 1;
       "MB_TCP_CLIENT".MB_Client_Sending_1.Input.MB_DATA_ADDR := 40017;
       "MB_TCP_CLIENT".MB_Client_Sending_1.Input.DATA_LEN := 13;
       "MB_TCP_CLIENT".MB_Client_Sending_1.Input.req := TRUE;
       "MB_TCP_CLIENT".MB_Client_Sending_1.tagsStep."step" := 2;
   END_IF;
END_REGION

REGION Network 4: Wysyłanie danych - step 2
   // poziom napełniania, opróżniania
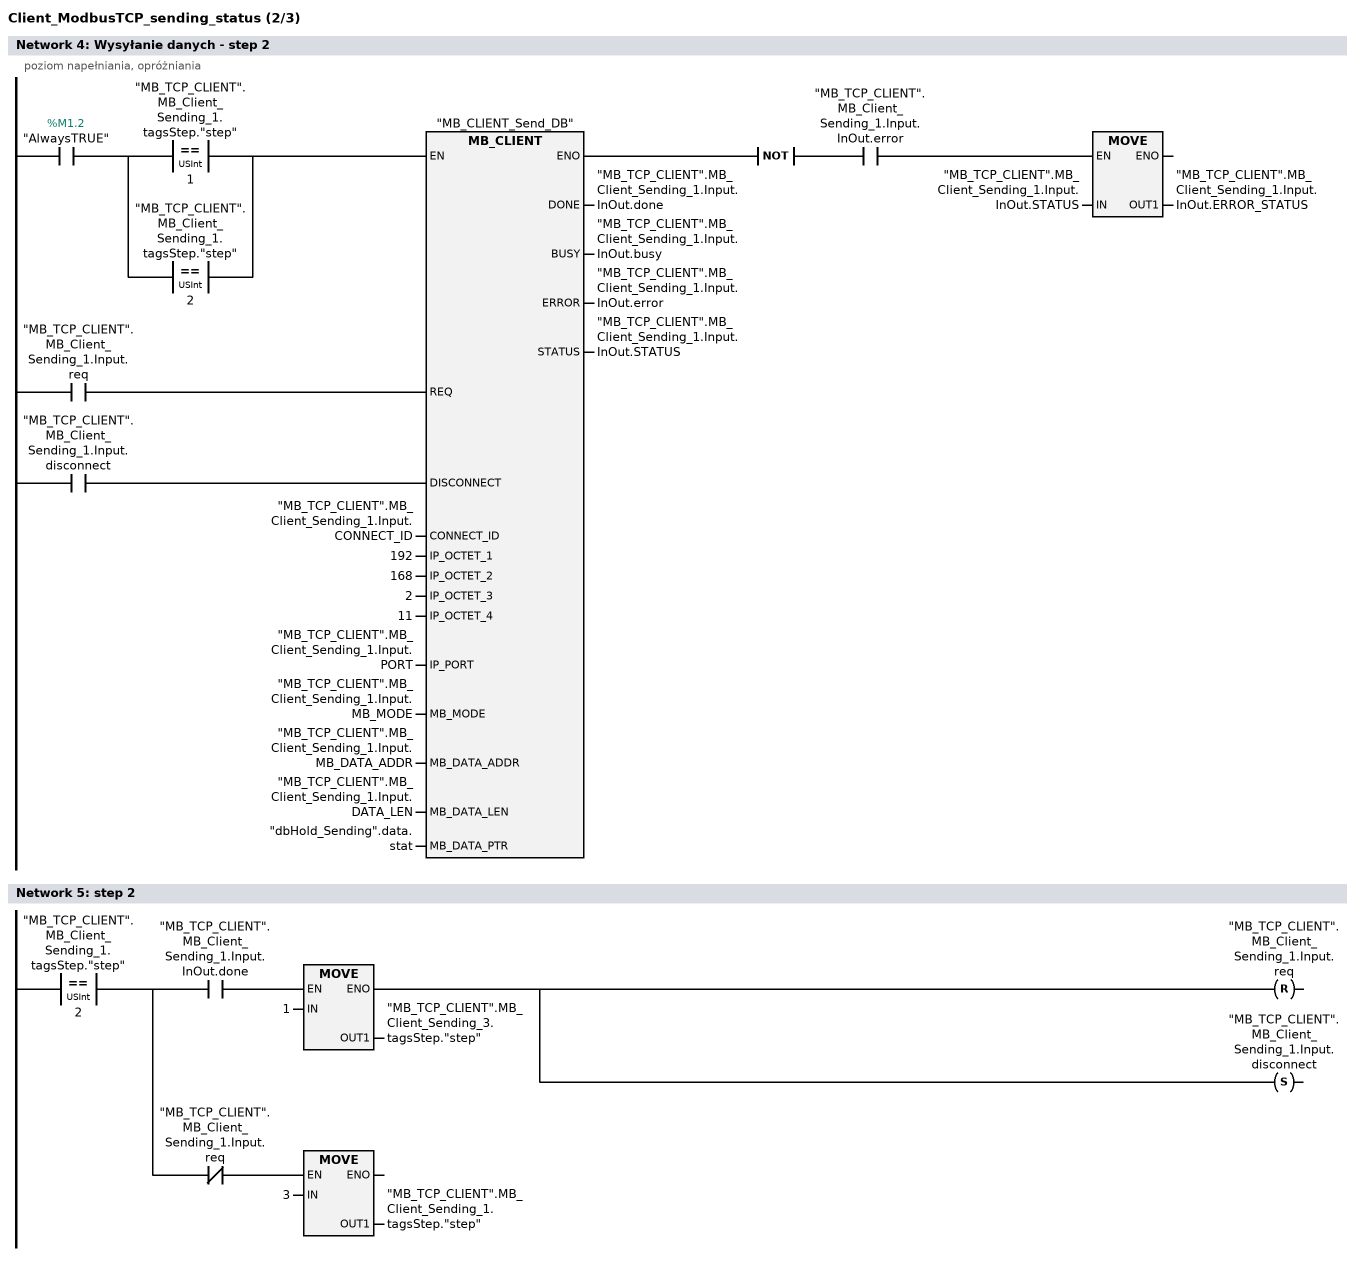
   RUNG wire#powerrail
      Contact( "AlwaysTRUE" )
      wire#w1
      { S7_Templates := "SrcType := USInt" } EQ_Contact(in1 := "MB_TCP_CLIENT".MB_Client_Sending_1.tagsStep."step", in2 := 1)
      wire#w2
      { S7_Templates := "[card1200 := 1, card1500 := 0]" } "MB_CLIENT_Send_DB".MB_CLIENT(REQ := wire#w3, DISCONNECT := wire#w4, CONNECT_ID := "MB_TCP_CLIENT".MB_Client_Sending_1.Input.CONNECT_ID, IP_OCTET_1 := 192, IP_OCTET_2 := 168, IP_OCTET_3 := 2, IP_OCTET_4 := 11, IP_PORT := "MB_TCP_CLIENT".MB_Client_Sending_1.Input.PORT, MB_MODE := "MB_TCP_CLIENT".MB_Client_Sending_1.Input.MB_MODE, MB_DATA_ADDR := "MB_TCP_CLIENT".MB_Client_Sending_1.Input.MB_DATA_ADDR, MB_DATA_LEN := "MB_TCP_CLIENT".MB_Client_Sending_1.Input.DATA_LEN, MB_DATA_PTR := "dbHold_Sending".data.stat, DONE => "MB_TCP_CLIENT".MB_Client_Sending_1.Input.InOut.done, BUSY => "MB_TCP_CLIENT".MB_Client_Sending_1.Input.InOut.busy, ERROR => "MB_TCP_CLIENT".MB_Client_Sending_1.Input.InOut.error, STATUS => "MB_TCP_CLIENT".MB_Client_Sending_1.Input.InOut.STATUS)
      Not()
      Contact( "MB_TCP_CLIENT".MB_Client_Sending_1.Input.InOut.error )
      Move(in := "MB_TCP_CLIENT".MB_Client_Sending_1.Input.InOut.STATUS, out1 => "MB_TCP_CLIENT".MB_Client_Sending_1.Input.InOut.ERROR_STATUS)
   END_RUNG
   RUNG wire#w1
      { S7_Templates := "SrcType := USInt" } EQ_Contact(in1 := "MB_TCP_CLIENT".MB_Client_Sending_1.tagsStep."step", in2 := 2)
   END_RUNG wire#w2
   RUNG wire#powerrail
      Contact( "MB_TCP_CLIENT".MB_Client_Sending_1.Input.req )
   END_RUNG wire#w3
   RUNG wire#powerrail
      Contact( "MB_TCP_CLIENT".MB_Client_Sending_1.Input.disconnect )
   END_RUNG wire#w4
   // the same network as SCL:
   #_w1 := "AlwaysTRUE" AND (("MB_TCP_CLIENT".MB_Client_Sending_1.tagsStep."step" = 1) OR ("MB_TCP_CLIENT".MB_Client_Sending_1.tagsStep."step" = 2));
   "MB_CLIENT_Send_DB"(EN := #_w1,   // MB_CLIENT
                       REQ := "MB_TCP_CLIENT".MB_Client_Sending_1.Input.req,
                       DISCONNECT := "MB_TCP_CLIENT".MB_Client_Sending_1.Input.disconnect,
                       CONNECT_ID := "MB_TCP_CLIENT".MB_Client_Sending_1.Input.CONNECT_ID,
                       IP_OCTET_1 := 192,
                       IP_OCTET_2 := 168,
                       IP_OCTET_3 := 2,
                       IP_OCTET_4 := 11,
                       IP_PORT := "MB_TCP_CLIENT".MB_Client_Sending_1.Input.PORT,
                       MB_MODE := "MB_TCP_CLIENT".MB_Client_Sending_1.Input.MB_MODE,
                       MB_DATA_ADDR := "MB_TCP_CLIENT".MB_Client_Sending_1.Input.MB_DATA_ADDR,
                       MB_DATA_LEN := "MB_TCP_CLIENT".MB_Client_Sending_1.Input.DATA_LEN,
                       MB_DATA_PTR := "dbHold_Sending".data.stat,
                       DONE => "MB_TCP_CLIENT".MB_Client_Sending_1.Input.InOut.done,
                       BUSY => "MB_TCP_CLIENT".MB_Client_Sending_1.Input.InOut.busy,
                       ERROR => "MB_TCP_CLIENT".MB_Client_Sending_1.Input.InOut.error,
                       STATUS => "MB_TCP_CLIENT".MB_Client_Sending_1.Input.InOut.STATUS,
                       ENO => #_w2);
   IF NOT #_w2 AND "MB_TCP_CLIENT".MB_Client_Sending_1.Input.InOut.error THEN
       "MB_TCP_CLIENT".MB_Client_Sending_1.Input.InOut.ERROR_STATUS := "MB_TCP_CLIENT".MB_Client_Sending_1.Input.InOut.STATUS;
   END_IF;
END_REGION

REGION Network 5: step 2
   RUNG wire#powerrail
      { S7_Templates := "SrcType := USInt" } EQ_Contact(in1 := "MB_TCP_CLIENT".MB_Client_Sending_1.tagsStep."step", in2 := 2)
      wire#w1
      Contact( "MB_TCP_CLIENT".MB_Client_Sending_1.Input.InOut.done )
      Move(in := 1, out1 => "MB_TCP_CLIENT".MB_Client_Sending_3.tagsStep."step")
      wire#w2
      R_Coil( "MB_TCP_CLIENT".MB_Client_Sending_1.Input.req )
   END_RUNG
   RUNG wire#w2
      S_Coil( "MB_TCP_CLIENT".MB_Client_Sending_1.Input.disconnect )
   END_RUNG
   RUNG wire#w1
      I_Contact( "MB_TCP_CLIENT".MB_Client_Sending_1.Input.req )
      Move(in := 3, out1 => "MB_TCP_CLIENT".MB_Client_Sending_1.tagsStep."step")
   END_RUNG
   // the same network as SCL:
   #_w1 := "MB_TCP_CLIENT".MB_Client_Sending_1.tagsStep."step" = 2;
   IF #_w1 AND "MB_TCP_CLIENT".MB_Client_Sending_1.Input.InOut.done THEN
       "MB_TCP_CLIENT".MB_Client_Sending_3.tagsStep."step" := 1;
       "MB_TCP_CLIENT".MB_Client_Sending_1.Input.req := FALSE;
       "MB_TCP_CLIENT".MB_Client_Sending_1.Input.disconnect := TRUE;
   END_IF;
   IF #_w1 AND NOT "MB_TCP_CLIENT".MB_Client_Sending_1.Input.req THEN
       "MB_TCP_CLIENT".MB_Client_Sending_1.tagsStep."step" := 3;
   END_IF;
END_REGION

REGION Network 6
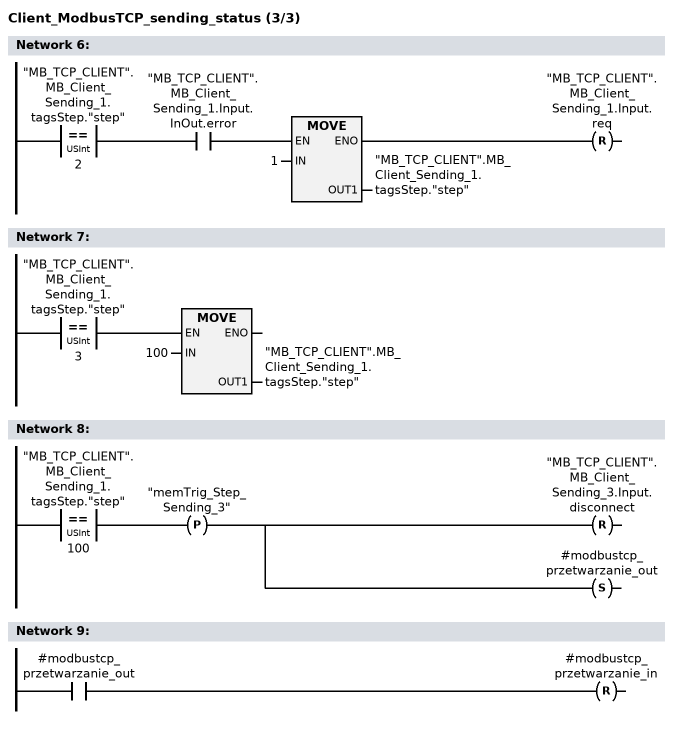
   RUNG wire#powerrail
      { S7_Templates := "SrcType := USInt" } EQ_Contact(in1 := "MB_TCP_CLIENT".MB_Client_Sending_1.tagsStep."step", in2 := 2)
      Contact( "MB_TCP_CLIENT".MB_Client_Sending_1.Input.InOut.error )
      Move(in := 1, out1 => "MB_TCP_CLIENT".MB_Client_Sending_1.tagsStep."step")
      R_Coil( "MB_TCP_CLIENT".MB_Client_Sending_1.Input.req )
   END_RUNG
   // the same network as SCL:
   #_w1 := ("MB_TCP_CLIENT".MB_Client_Sending_1.tagsStep."step" = 2) AND "MB_TCP_CLIENT".MB_Client_Sending_1.Input.InOut.error;
   IF #_w1 THEN
       "MB_TCP_CLIENT".MB_Client_Sending_1.tagsStep."step" := 1;
       "MB_TCP_CLIENT".MB_Client_Sending_1.Input.req := FALSE;
   END_IF;
END_REGION

REGION Network 7
   RUNG wire#powerrail
      { S7_Templates := "SrcType := USInt" } EQ_Contact(in1 := "MB_TCP_CLIENT".MB_Client_Sending_1.tagsStep."step", in2 := 3)
      Move(in := 100, out1 => "MB_TCP_CLIENT".MB_Client_Sending_1.tagsStep."step")
   END_RUNG
   // the same network as SCL:
   IF "MB_TCP_CLIENT".MB_Client_Sending_1.tagsStep."step" = 3 THEN
       "MB_TCP_CLIENT".MB_Client_Sending_1.tagsStep."step" := 100;
   END_IF;
END_REGION

REGION Network 8
   RUNG wire#powerrail
      { S7_Templates := "SrcType := USInt" } EQ_Contact(in1 := "MB_TCP_CLIENT".MB_Client_Sending_1.tagsStep."step", in2 := 100)
      P_Trig( "memTrig_Step_Sending_3" )
      wire#w1
      R_Coil( "MB_TCP_CLIENT".MB_Client_Sending_3.Input.disconnect )
   END_RUNG
   RUNG wire#w1
      S_Coil( #modbustcp_przetwarzanie_out )
   END_RUNG
   // the same network as SCL:
   #_w1 := "MB_TCP_CLIENT".MB_Client_Sending_1.tagsStep."step" = 100;
   #_w2 := #_w1 AND NOT "memTrig_Step_Sending_3";   // rising edge
   "memTrig_Step_Sending_3" := #_w1;
   IF #_w2 THEN
       "MB_TCP_CLIENT".MB_Client_Sending_3.Input.disconnect := FALSE;
       #modbustcp_przetwarzanie_out := TRUE;
   END_IF;
END_REGION

REGION Network 9
   RUNG wire#powerrail
      Contact( #modbustcp_przetwarzanie_out )
      R_Coil( #modbustcp_przetwarzanie_in )
   END_RUNG
   // the same network as SCL:
   IF #modbustcp_przetwarzanie_out THEN #modbustcp_przetwarzanie_in := FALSE; END_IF;
END_REGION
END_FUNCTION_BLOCK

FUNCTION_BLOCK "Client_ModbusTCP_sending_parameters"   // FB13, LAD
TITLE = Przesłanie parametrów sterowania
{ S7_Optimized_Access := 'TRUE' }
AUTHOR : rtecmer
VERSION : 0.1
// funkcja przkazuje parametry sterowania do PLC 1
// stored: AutoNumber true, IsIECCheckEnabled false, IsRetainMemResEnabled false, MemoryReserve 250, SetENOAutomatically false, UDAEnableTagReadback false
   VAR_IN_OUT
      modbustcp_przetwarzanie_in : Bool;
      modbustcp_przetwarzanie_out : Bool;
   END_VAR
   VAR_TEMP   // added for the SCL form of the ladder/FBD networks
      _w1 : Bool;
      _w2 : Bool;
   END_VAR
BEGIN

REGION Network 1: Inicjacja modbus po błędzie i restarcie
END_REGION

REGION Network 2
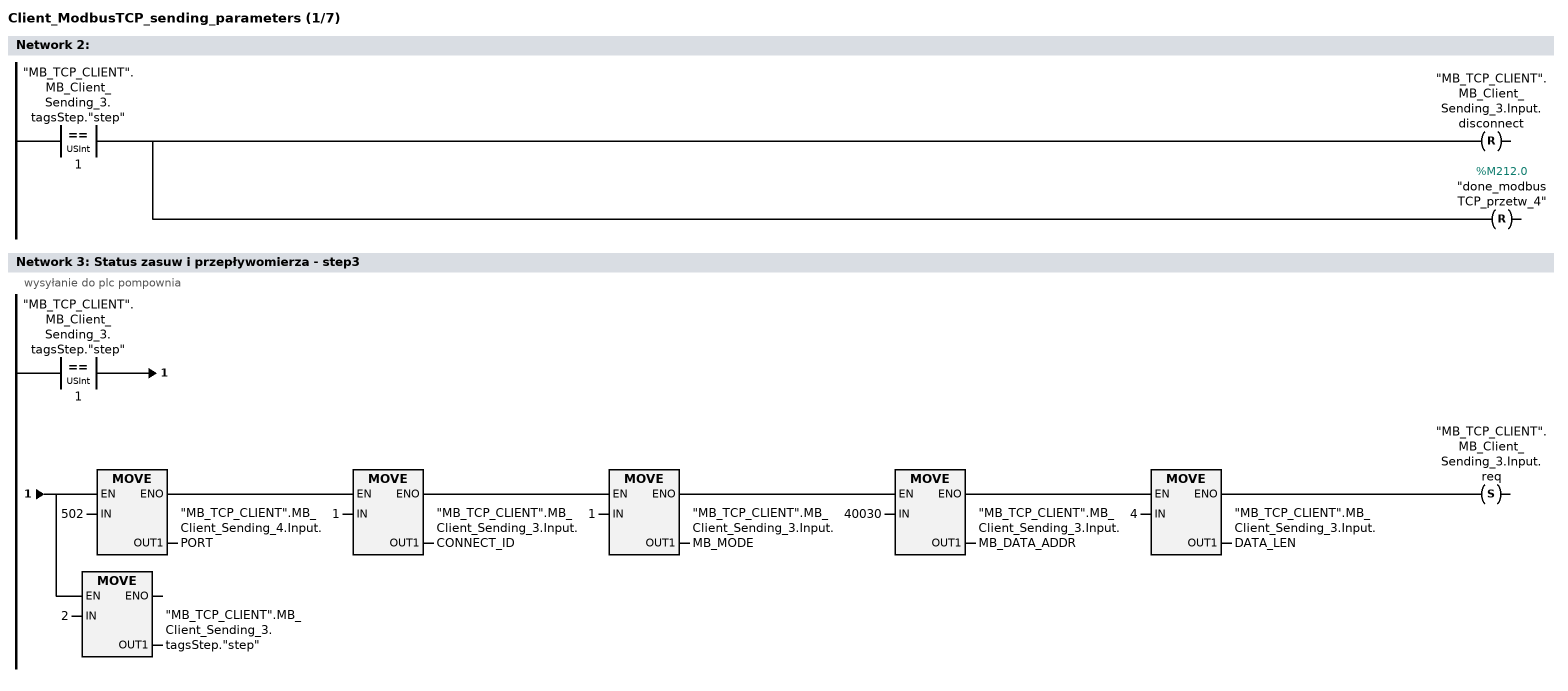
   RUNG wire#powerrail
      { S7_Templates := "SrcType := USInt" } EQ_Contact(in1 := "MB_TCP_CLIENT".MB_Client_Sending_3.tagsStep."step", in2 := 1)
      wire#w1
      R_Coil( "MB_TCP_CLIENT".MB_Client_Sending_3.Input.disconnect )
   END_RUNG
   RUNG wire#w1
      R_Coil( "done_modbusTCP_przetw_4" )
   END_RUNG
   // the same network as SCL:
   IF "MB_TCP_CLIENT".MB_Client_Sending_3.tagsStep."step" = 1 THEN
       "MB_TCP_CLIENT".MB_Client_Sending_3.Input.disconnect := FALSE;
       "done_modbusTCP_przetw_4" := FALSE;
   END_IF;
END_REGION

REGION Network 3: Status zasuw i przepływomierza - step3
   // wysyłanie do plc pompownia
   RUNG wire#powerrail
      { S7_Templates := "SrcType := USInt" } EQ_Contact(in1 := "MB_TCP_CLIENT".MB_Client_Sending_3.tagsStep."step", in2 := 1)
      wire#w1
      { S7_GenerateENO := "TRUE" } Move(in := 502, out1 => "MB_TCP_CLIENT".MB_Client_Sending_4.Input.PORT)
      { S7_GenerateENO := "TRUE" } Move(in := 1, out1 => "MB_TCP_CLIENT".MB_Client_Sending_3.Input.CONNECT_ID)
      { S7_GenerateENO := "TRUE" } Move(in := 1, out1 => "MB_TCP_CLIENT".MB_Client_Sending_3.Input.MB_MODE)
      { S7_GenerateENO := "TRUE" } Move(in := 40030, out1 => "MB_TCP_CLIENT".MB_Client_Sending_3.Input.MB_DATA_ADDR)
      { S7_GenerateENO := "TRUE" } Move(in := 4, out1 => "MB_TCP_CLIENT".MB_Client_Sending_3.Input.DATA_LEN)
      S_Coil( "MB_TCP_CLIENT".MB_Client_Sending_3.Input.req )
   END_RUNG
   RUNG wire#w1
      { S7_GenerateENO := "TRUE" } Move(in := 2, out1 => "MB_TCP_CLIENT".MB_Client_Sending_3.tagsStep."step")
   END_RUNG
   // the same network as SCL:
   // ENO of a box is taken as its EN; it also drops when the box reports an error
   IF "MB_TCP_CLIENT".MB_Client_Sending_3.tagsStep."step" = 1 THEN
       "MB_TCP_CLIENT".MB_Client_Sending_4.Input.PORT := 502;
       "MB_TCP_CLIENT".MB_Client_Sending_3.Input.CONNECT_ID := 1;
       "MB_TCP_CLIENT".MB_Client_Sending_3.Input.MB_MODE := 1;
       "MB_TCP_CLIENT".MB_Client_Sending_3.Input.MB_DATA_ADDR := 40030;
       "MB_TCP_CLIENT".MB_Client_Sending_3.Input.DATA_LEN := 4;
       "MB_TCP_CLIENT".MB_Client_Sending_3.Input.req := TRUE;
       "MB_TCP_CLIENT".MB_Client_Sending_3.tagsStep."step" := 2;
   END_IF;
END_REGION

REGION Network 4: Wysyłanie danych - step 2
   // poziom napełniania, opróżniania
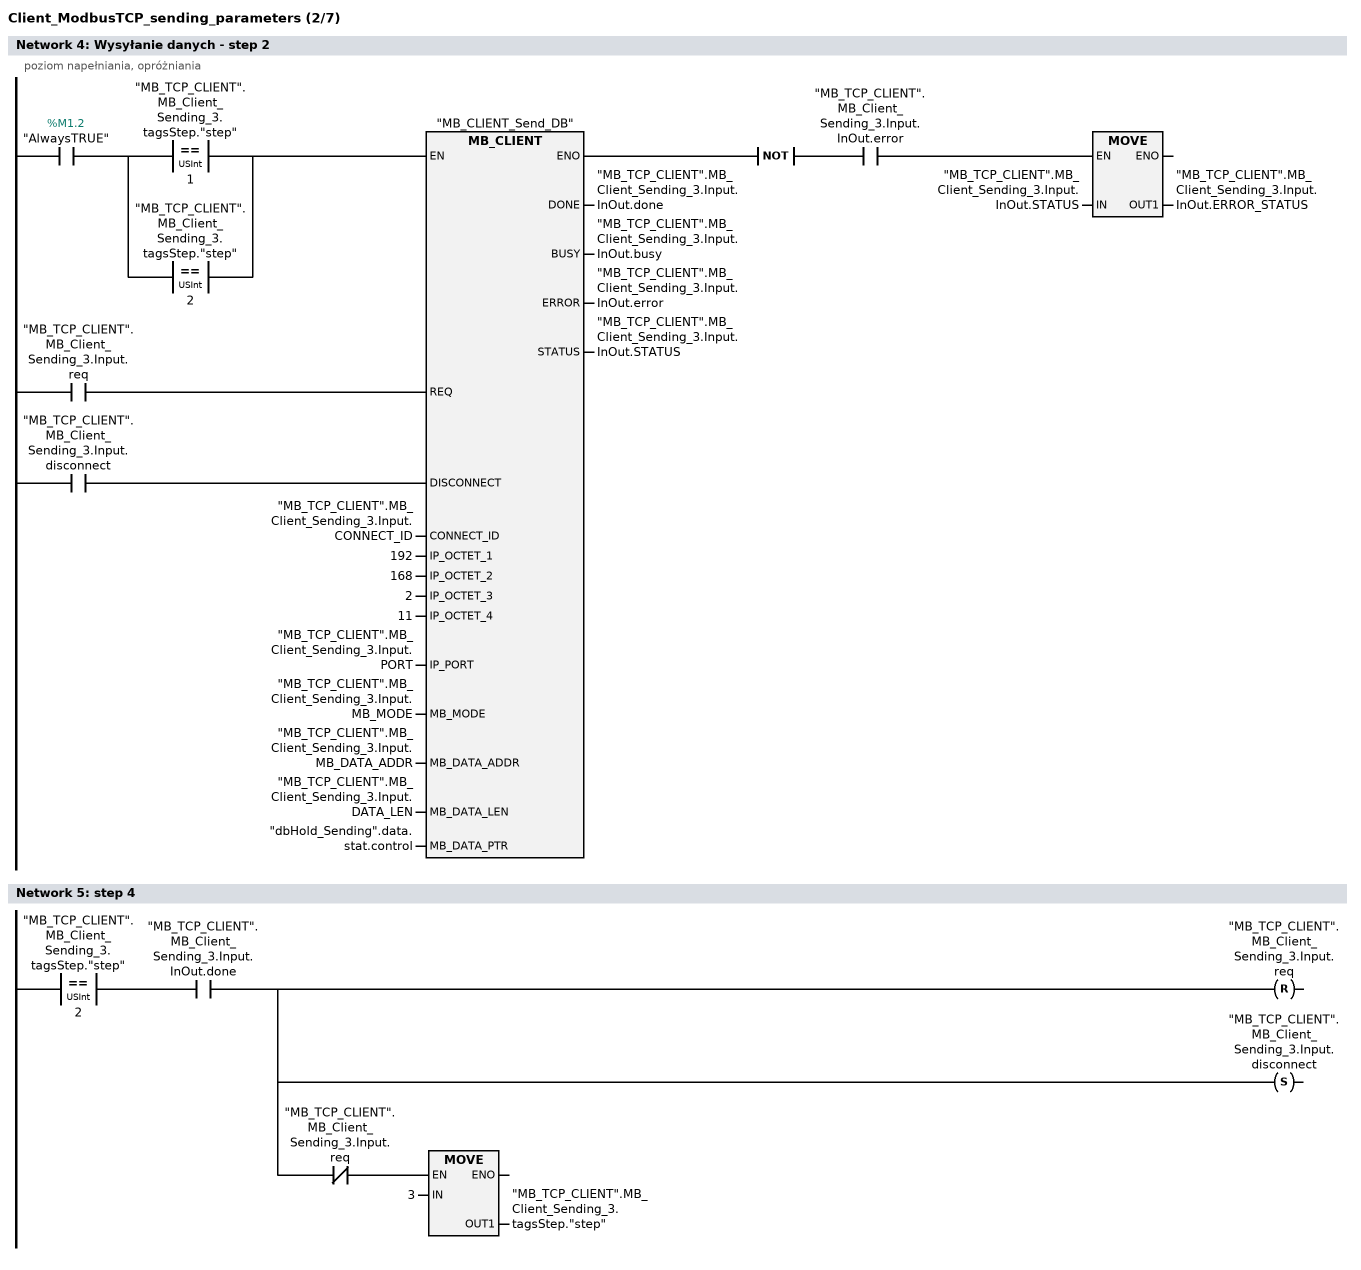
   RUNG wire#powerrail
      Contact( "AlwaysTRUE" )
      wire#w1
      { S7_Templates := "SrcType := USInt" } EQ_Contact(in1 := "MB_TCP_CLIENT".MB_Client_Sending_3.tagsStep."step", in2 := 1)
      wire#w2
      { S7_Templates := "[card1200 := 1, card1500 := 0]" } "MB_CLIENT_Send_DB".MB_CLIENT(REQ := wire#w3, DISCONNECT := wire#w4, CONNECT_ID := "MB_TCP_CLIENT".MB_Client_Sending_3.Input.CONNECT_ID, IP_OCTET_1 := 192, IP_OCTET_2 := 168, IP_OCTET_3 := 2, IP_OCTET_4 := 11, IP_PORT := "MB_TCP_CLIENT".MB_Client_Sending_3.Input.PORT, MB_MODE := "MB_TCP_CLIENT".MB_Client_Sending_3.Input.MB_MODE, MB_DATA_ADDR := "MB_TCP_CLIENT".MB_Client_Sending_3.Input.MB_DATA_ADDR, MB_DATA_LEN := "MB_TCP_CLIENT".MB_Client_Sending_3.Input.DATA_LEN, MB_DATA_PTR := "dbHold_Sending".data.stat.control, DONE => "MB_TCP_CLIENT".MB_Client_Sending_3.Input.InOut.done, BUSY => "MB_TCP_CLIENT".MB_Client_Sending_3.Input.InOut.busy, ERROR => "MB_TCP_CLIENT".MB_Client_Sending_3.Input.InOut.error, STATUS => "MB_TCP_CLIENT".MB_Client_Sending_3.Input.InOut.STATUS)
      Not()
      Contact( "MB_TCP_CLIENT".MB_Client_Sending_3.Input.InOut.error )
      Move(in := "MB_TCP_CLIENT".MB_Client_Sending_3.Input.InOut.STATUS, out1 => "MB_TCP_CLIENT".MB_Client_Sending_3.Input.InOut.ERROR_STATUS)
   END_RUNG
   RUNG wire#w1
      { S7_Templates := "SrcType := USInt" } EQ_Contact(in1 := "MB_TCP_CLIENT".MB_Client_Sending_3.tagsStep."step", in2 := 2)
   END_RUNG wire#w2
   RUNG wire#powerrail
      Contact( "MB_TCP_CLIENT".MB_Client_Sending_3.Input.req )
   END_RUNG wire#w3
   RUNG wire#powerrail
      Contact( "MB_TCP_CLIENT".MB_Client_Sending_3.Input.disconnect )
   END_RUNG wire#w4
   // the same network as SCL:
   #_w1 := "AlwaysTRUE" AND (("MB_TCP_CLIENT".MB_Client_Sending_3.tagsStep."step" = 1) OR ("MB_TCP_CLIENT".MB_Client_Sending_3.tagsStep."step" = 2));
   "MB_CLIENT_Send_DB"(EN := #_w1,   // MB_CLIENT
                       REQ := "MB_TCP_CLIENT".MB_Client_Sending_3.Input.req,
                       DISCONNECT := "MB_TCP_CLIENT".MB_Client_Sending_3.Input.disconnect,
                       CONNECT_ID := "MB_TCP_CLIENT".MB_Client_Sending_3.Input.CONNECT_ID,
                       IP_OCTET_1 := 192,
                       IP_OCTET_2 := 168,
                       IP_OCTET_3 := 2,
                       IP_OCTET_4 := 11,
                       IP_PORT := "MB_TCP_CLIENT".MB_Client_Sending_3.Input.PORT,
                       MB_MODE := "MB_TCP_CLIENT".MB_Client_Sending_3.Input.MB_MODE,
                       MB_DATA_ADDR := "MB_TCP_CLIENT".MB_Client_Sending_3.Input.MB_DATA_ADDR,
                       MB_DATA_LEN := "MB_TCP_CLIENT".MB_Client_Sending_3.Input.DATA_LEN,
                       MB_DATA_PTR := "dbHold_Sending".data.stat.control,
                       DONE => "MB_TCP_CLIENT".MB_Client_Sending_3.Input.InOut.done,
                       BUSY => "MB_TCP_CLIENT".MB_Client_Sending_3.Input.InOut.busy,
                       ERROR => "MB_TCP_CLIENT".MB_Client_Sending_3.Input.InOut.error,
                       STATUS => "MB_TCP_CLIENT".MB_Client_Sending_3.Input.InOut.STATUS,
                       ENO => #_w2);
   IF NOT #_w2 AND "MB_TCP_CLIENT".MB_Client_Sending_3.Input.InOut.error THEN
       "MB_TCP_CLIENT".MB_Client_Sending_3.Input.InOut.ERROR_STATUS := "MB_TCP_CLIENT".MB_Client_Sending_3.Input.InOut.STATUS;
   END_IF;
END_REGION

REGION Network 5: step 4
   RUNG wire#powerrail
      { S7_Templates := "SrcType := USInt" } EQ_Contact(in1 := "MB_TCP_CLIENT".MB_Client_Sending_3.tagsStep."step", in2 := 2)
      Contact( "MB_TCP_CLIENT".MB_Client_Sending_3.Input.InOut.done )
      wire#w1
      R_Coil( "MB_TCP_CLIENT".MB_Client_Sending_3.Input.req )
   END_RUNG
   RUNG wire#w1
      S_Coil( "MB_TCP_CLIENT".MB_Client_Sending_3.Input.disconnect )
   END_RUNG
   RUNG wire#w1
      I_Contact( "MB_TCP_CLIENT".MB_Client_Sending_3.Input.req )
      Move(in := 3, out1 => "MB_TCP_CLIENT".MB_Client_Sending_3.tagsStep."step")
   END_RUNG
   // the same network as SCL:
   #_w1 := ("MB_TCP_CLIENT".MB_Client_Sending_3.tagsStep."step" = 2) AND "MB_TCP_CLIENT".MB_Client_Sending_3.Input.InOut.done;
   IF #_w1 THEN
       "MB_TCP_CLIENT".MB_Client_Sending_3.Input.req := FALSE;
       "MB_TCP_CLIENT".MB_Client_Sending_3.Input.disconnect := TRUE;
   END_IF;
   IF #_w1 AND NOT "MB_TCP_CLIENT".MB_Client_Sending_3.Input.req THEN
       "MB_TCP_CLIENT".MB_Client_Sending_3.tagsStep."step" := 3;
   END_IF;
END_REGION

REGION Network 6
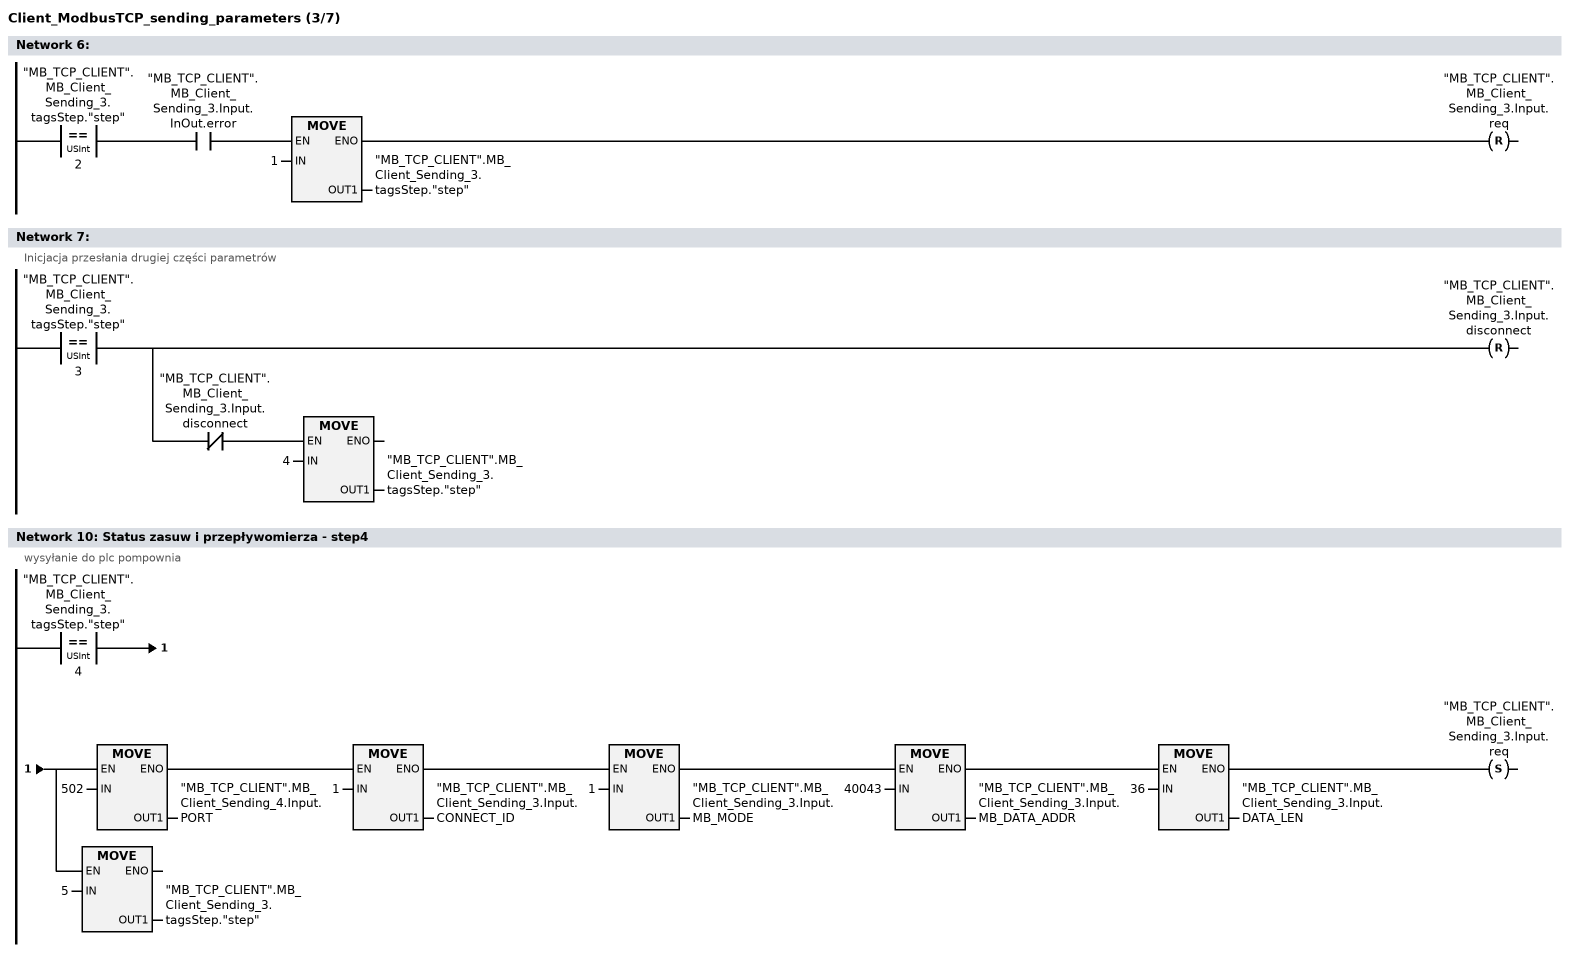
   RUNG wire#powerrail
      { S7_Templates := "SrcType := USInt" } EQ_Contact(in1 := "MB_TCP_CLIENT".MB_Client_Sending_3.tagsStep."step", in2 := 2)
      Contact( "MB_TCP_CLIENT".MB_Client_Sending_3.Input.InOut.error )
      Move(in := 1, out1 => "MB_TCP_CLIENT".MB_Client_Sending_3.tagsStep."step")
      R_Coil( "MB_TCP_CLIENT".MB_Client_Sending_3.Input.req )
   END_RUNG
   // the same network as SCL:
   #_w1 := ("MB_TCP_CLIENT".MB_Client_Sending_3.tagsStep."step" = 2) AND "MB_TCP_CLIENT".MB_Client_Sending_3.Input.InOut.error;
   IF #_w1 THEN
       "MB_TCP_CLIENT".MB_Client_Sending_3.tagsStep."step" := 1;
       "MB_TCP_CLIENT".MB_Client_Sending_3.Input.req := FALSE;
   END_IF;
END_REGION

REGION Network 7
   // Inicjacja przesłania drugiej części parametrów
   RUNG wire#powerrail
      { S7_Templates := "SrcType := USInt" } EQ_Contact(in1 := "MB_TCP_CLIENT".MB_Client_Sending_3.tagsStep."step", in2 := 3)
      wire#w1
      R_Coil( "MB_TCP_CLIENT".MB_Client_Sending_3.Input.disconnect )
   END_RUNG
   RUNG wire#w1
      I_Contact( "MB_TCP_CLIENT".MB_Client_Sending_3.Input.disconnect )
      Move(in := 4, out1 => "MB_TCP_CLIENT".MB_Client_Sending_3.tagsStep."step")
   END_RUNG
   // the same network as SCL:
   #_w1 := "MB_TCP_CLIENT".MB_Client_Sending_3.tagsStep."step" = 3;
   IF #_w1 THEN "MB_TCP_CLIENT".MB_Client_Sending_3.Input.disconnect := FALSE; END_IF;
   IF #_w1 AND NOT "MB_TCP_CLIENT".MB_Client_Sending_3.Input.disconnect THEN
       "MB_TCP_CLIENT".MB_Client_Sending_3.tagsStep."step" := 4;
   END_IF;
END_REGION

REGION Network 10: Status zasuw i przepływomierza - step4
   // wysyłanie do plc pompownia
   RUNG wire#powerrail
      { S7_Templates := "SrcType := USInt" } EQ_Contact(in1 := "MB_TCP_CLIENT".MB_Client_Sending_3.tagsStep."step", in2 := 4)
      wire#w1
      { S7_GenerateENO := "TRUE" } Move(in := 502, out1 => "MB_TCP_CLIENT".MB_Client_Sending_4.Input.PORT)
      { S7_GenerateENO := "TRUE" } Move(in := 1, out1 => "MB_TCP_CLIENT".MB_Client_Sending_3.Input.CONNECT_ID)
      { S7_GenerateENO := "TRUE" } Move(in := 1, out1 => "MB_TCP_CLIENT".MB_Client_Sending_3.Input.MB_MODE)
      { S7_GenerateENO := "TRUE" } Move(in := 40043, out1 => "MB_TCP_CLIENT".MB_Client_Sending_3.Input.MB_DATA_ADDR)
      { S7_GenerateENO := "TRUE" } Move(in := 36, out1 => "MB_TCP_CLIENT".MB_Client_Sending_3.Input.DATA_LEN)
      S_Coil( "MB_TCP_CLIENT".MB_Client_Sending_3.Input.req )
   END_RUNG
   RUNG wire#w1
      { S7_GenerateENO := "TRUE" } Move(in := 5, out1 => "MB_TCP_CLIENT".MB_Client_Sending_3.tagsStep."step")
   END_RUNG
   // the same network as SCL:
   // ENO of a box is taken as its EN; it also drops when the box reports an error
   IF "MB_TCP_CLIENT".MB_Client_Sending_3.tagsStep."step" = 4 THEN
       "MB_TCP_CLIENT".MB_Client_Sending_4.Input.PORT := 502;
       "MB_TCP_CLIENT".MB_Client_Sending_3.Input.CONNECT_ID := 1;
       "MB_TCP_CLIENT".MB_Client_Sending_3.Input.MB_MODE := 1;
       "MB_TCP_CLIENT".MB_Client_Sending_3.Input.MB_DATA_ADDR := 40043;
       "MB_TCP_CLIENT".MB_Client_Sending_3.Input.DATA_LEN := 36;
       "MB_TCP_CLIENT".MB_Client_Sending_3.Input.req := TRUE;
       "MB_TCP_CLIENT".MB_Client_Sending_3.tagsStep."step" := 5;
   END_IF;
END_REGION

REGION Network 11: Wysyłanie danych - step 2
   // poziom napełniania, opróżniania
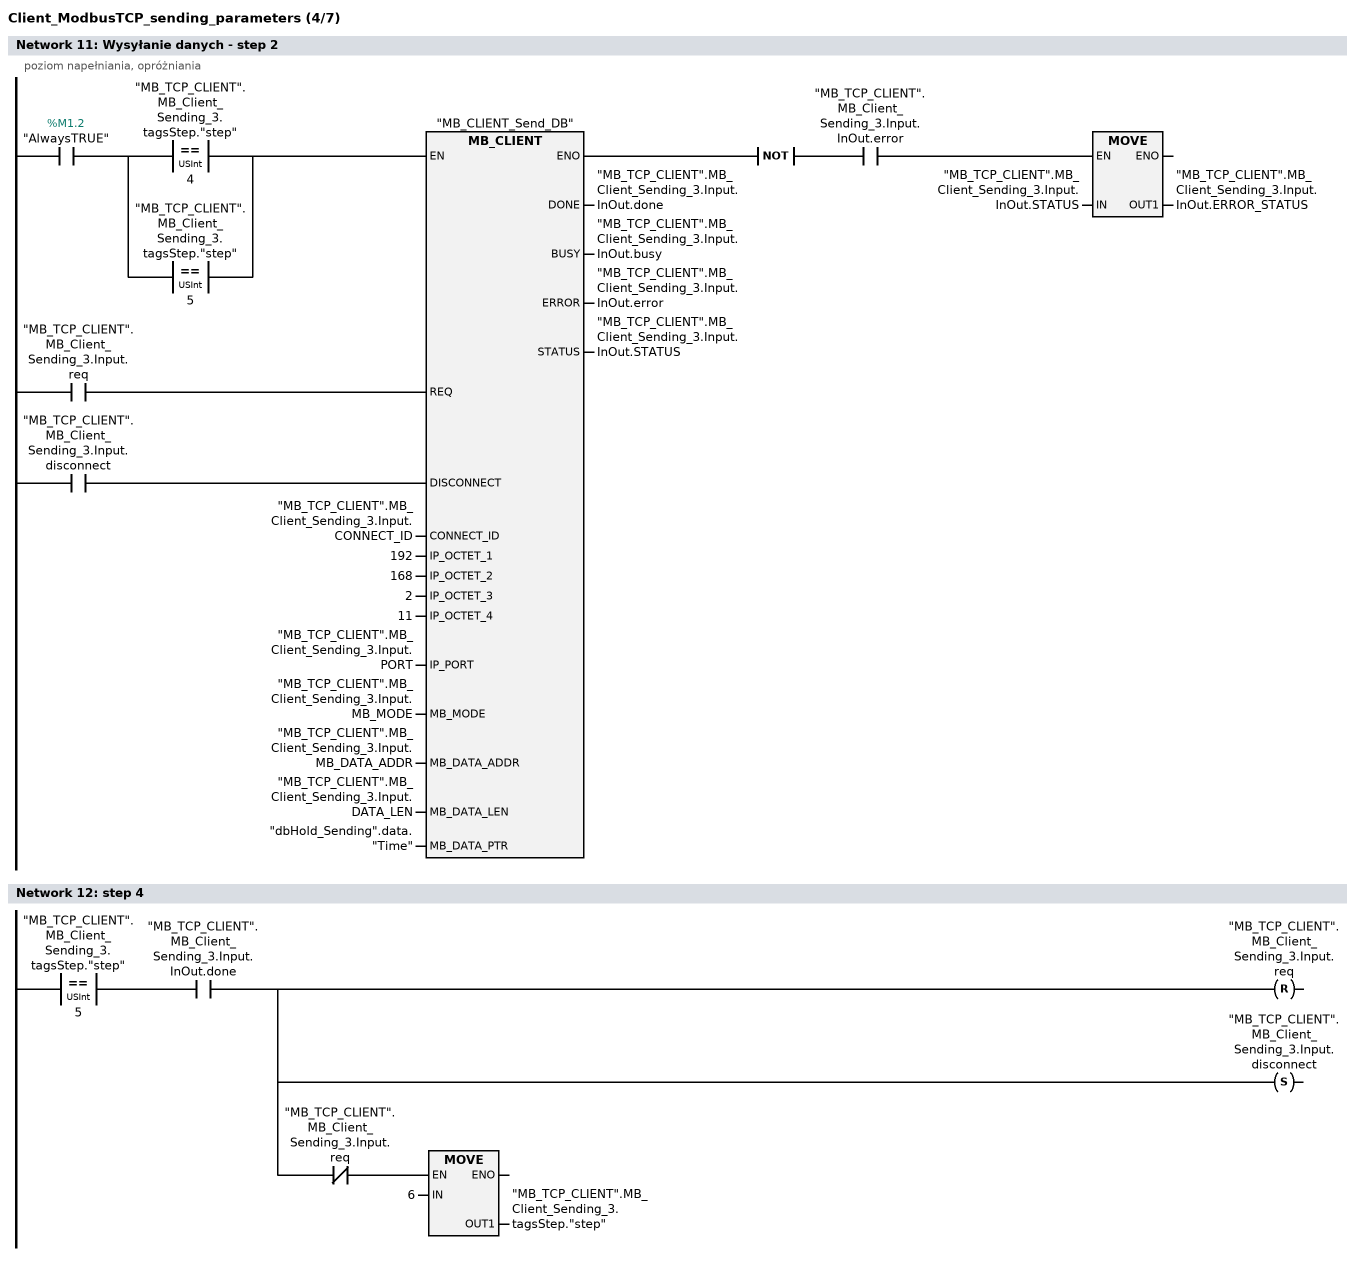
   RUNG wire#powerrail
      Contact( "AlwaysTRUE" )
      wire#w1
      { S7_Templates := "SrcType := USInt" } EQ_Contact(in1 := "MB_TCP_CLIENT".MB_Client_Sending_3.tagsStep."step", in2 := 4)
      wire#w2
      { S7_Templates := "[card1200 := 1, card1500 := 0]" } "MB_CLIENT_Send_DB".MB_CLIENT(REQ := wire#w3, DISCONNECT := wire#w4, CONNECT_ID := "MB_TCP_CLIENT".MB_Client_Sending_3.Input.CONNECT_ID, IP_OCTET_1 := 192, IP_OCTET_2 := 168, IP_OCTET_3 := 2, IP_OCTET_4 := 11, IP_PORT := "MB_TCP_CLIENT".MB_Client_Sending_3.Input.PORT, MB_MODE := "MB_TCP_CLIENT".MB_Client_Sending_3.Input.MB_MODE, MB_DATA_ADDR := "MB_TCP_CLIENT".MB_Client_Sending_3.Input.MB_DATA_ADDR, MB_DATA_LEN := "MB_TCP_CLIENT".MB_Client_Sending_3.Input.DATA_LEN, MB_DATA_PTR := "dbHold_Sending".data."Time", DONE => "MB_TCP_CLIENT".MB_Client_Sending_3.Input.InOut.done, BUSY => "MB_TCP_CLIENT".MB_Client_Sending_3.Input.InOut.busy, ERROR => "MB_TCP_CLIENT".MB_Client_Sending_3.Input.InOut.error, STATUS => "MB_TCP_CLIENT".MB_Client_Sending_3.Input.InOut.STATUS)
      Not()
      Contact( "MB_TCP_CLIENT".MB_Client_Sending_3.Input.InOut.error )
      Move(in := "MB_TCP_CLIENT".MB_Client_Sending_3.Input.InOut.STATUS, out1 => "MB_TCP_CLIENT".MB_Client_Sending_3.Input.InOut.ERROR_STATUS)
   END_RUNG
   RUNG wire#w1
      { S7_Templates := "SrcType := USInt" } EQ_Contact(in1 := "MB_TCP_CLIENT".MB_Client_Sending_3.tagsStep."step", in2 := 5)
   END_RUNG wire#w2
   RUNG wire#powerrail
      Contact( "MB_TCP_CLIENT".MB_Client_Sending_3.Input.req )
   END_RUNG wire#w3
   RUNG wire#powerrail
      Contact( "MB_TCP_CLIENT".MB_Client_Sending_3.Input.disconnect )
   END_RUNG wire#w4
   // the same network as SCL:
   #_w1 := "AlwaysTRUE" AND (("MB_TCP_CLIENT".MB_Client_Sending_3.tagsStep."step" = 4) OR ("MB_TCP_CLIENT".MB_Client_Sending_3.tagsStep."step" = 5));
   "MB_CLIENT_Send_DB"(EN := #_w1,   // MB_CLIENT
                       REQ := "MB_TCP_CLIENT".MB_Client_Sending_3.Input.req,
                       DISCONNECT := "MB_TCP_CLIENT".MB_Client_Sending_3.Input.disconnect,
                       CONNECT_ID := "MB_TCP_CLIENT".MB_Client_Sending_3.Input.CONNECT_ID,
                       IP_OCTET_1 := 192,
                       IP_OCTET_2 := 168,
                       IP_OCTET_3 := 2,
                       IP_OCTET_4 := 11,
                       IP_PORT := "MB_TCP_CLIENT".MB_Client_Sending_3.Input.PORT,
                       MB_MODE := "MB_TCP_CLIENT".MB_Client_Sending_3.Input.MB_MODE,
                       MB_DATA_ADDR := "MB_TCP_CLIENT".MB_Client_Sending_3.Input.MB_DATA_ADDR,
                       MB_DATA_LEN := "MB_TCP_CLIENT".MB_Client_Sending_3.Input.DATA_LEN,
                       MB_DATA_PTR := "dbHold_Sending".data."Time",
                       DONE => "MB_TCP_CLIENT".MB_Client_Sending_3.Input.InOut.done,
                       BUSY => "MB_TCP_CLIENT".MB_Client_Sending_3.Input.InOut.busy,
                       ERROR => "MB_TCP_CLIENT".MB_Client_Sending_3.Input.InOut.error,
                       STATUS => "MB_TCP_CLIENT".MB_Client_Sending_3.Input.InOut.STATUS,
                       ENO => #_w2);
   IF NOT #_w2 AND "MB_TCP_CLIENT".MB_Client_Sending_3.Input.InOut.error THEN
       "MB_TCP_CLIENT".MB_Client_Sending_3.Input.InOut.ERROR_STATUS := "MB_TCP_CLIENT".MB_Client_Sending_3.Input.InOut.STATUS;
   END_IF;
END_REGION

REGION Network 12: step 4
   RUNG wire#powerrail
      { S7_Templates := "SrcType := USInt" } EQ_Contact(in1 := "MB_TCP_CLIENT".MB_Client_Sending_3.tagsStep."step", in2 := 5)
      Contact( "MB_TCP_CLIENT".MB_Client_Sending_3.Input.InOut.done )
      wire#w1
      R_Coil( "MB_TCP_CLIENT".MB_Client_Sending_3.Input.req )
   END_RUNG
   RUNG wire#w1
      S_Coil( "MB_TCP_CLIENT".MB_Client_Sending_3.Input.disconnect )
   END_RUNG
   RUNG wire#w1
      I_Contact( "MB_TCP_CLIENT".MB_Client_Sending_3.Input.req )
      Move(in := 6, out1 => "MB_TCP_CLIENT".MB_Client_Sending_3.tagsStep."step")
   END_RUNG
   // the same network as SCL:
   #_w1 := ("MB_TCP_CLIENT".MB_Client_Sending_3.tagsStep."step" = 5) AND "MB_TCP_CLIENT".MB_Client_Sending_3.Input.InOut.done;
   IF #_w1 THEN
       "MB_TCP_CLIENT".MB_Client_Sending_3.Input.req := FALSE;
       "MB_TCP_CLIENT".MB_Client_Sending_3.Input.disconnect := TRUE;
   END_IF;
   IF #_w1 AND NOT "MB_TCP_CLIENT".MB_Client_Sending_3.Input.req THEN
       "MB_TCP_CLIENT".MB_Client_Sending_3.tagsStep."step" := 6;
   END_IF;
END_REGION

REGION Network 13
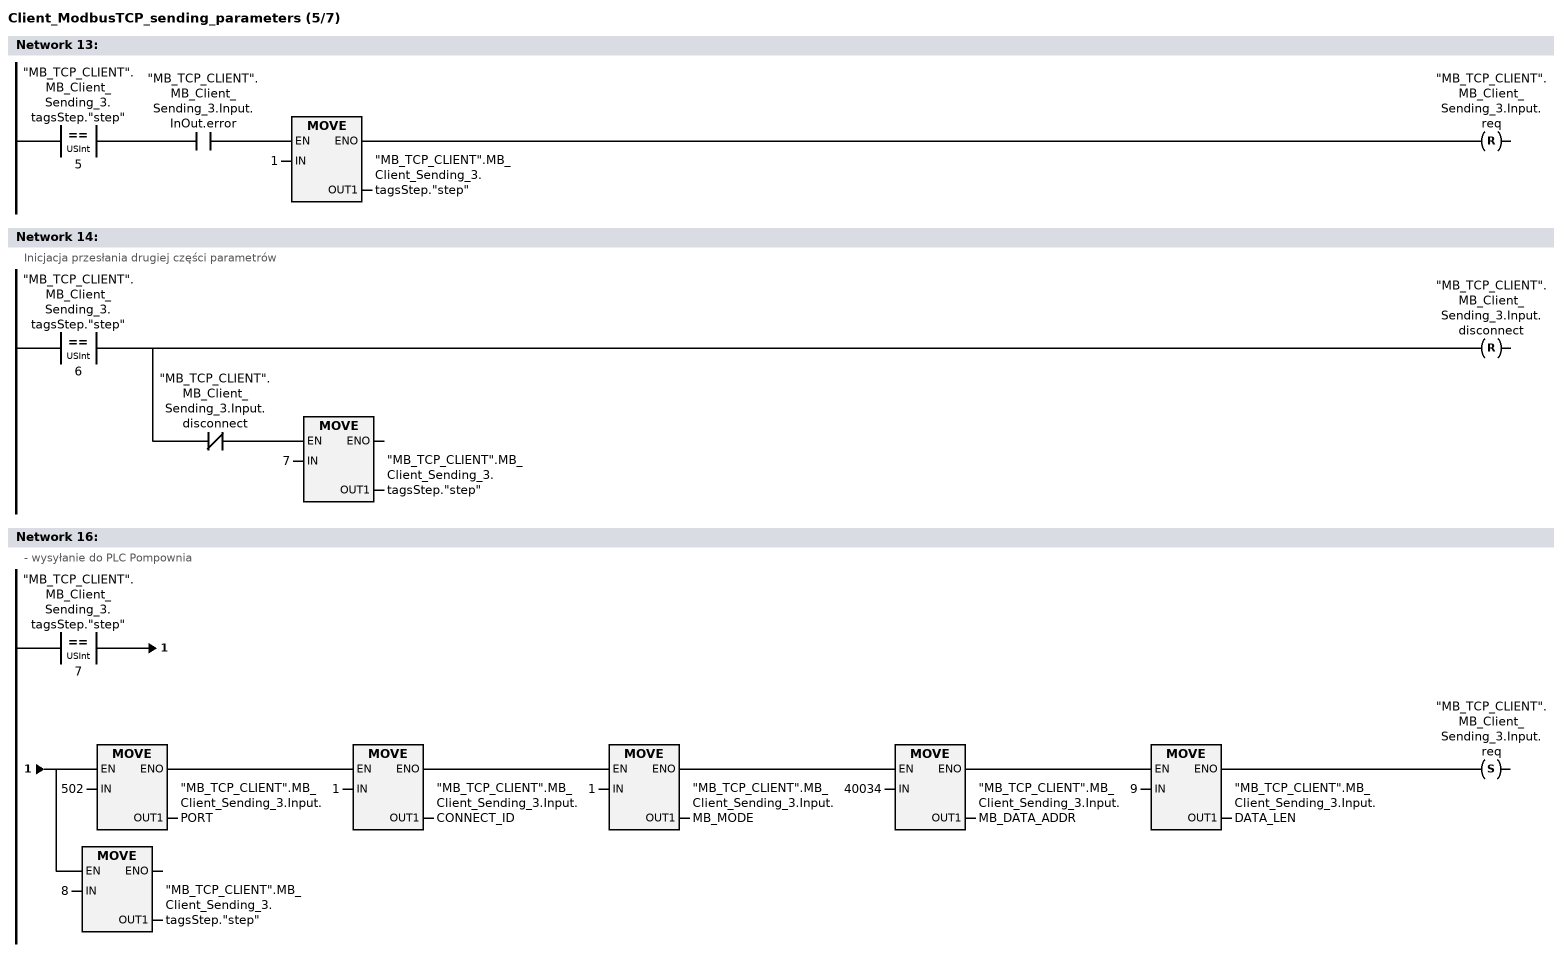
   RUNG wire#powerrail
      { S7_Templates := "SrcType := USInt" } EQ_Contact(in1 := "MB_TCP_CLIENT".MB_Client_Sending_3.tagsStep."step", in2 := 5)
      Contact( "MB_TCP_CLIENT".MB_Client_Sending_3.Input.InOut.error )
      Move(in := 1, out1 => "MB_TCP_CLIENT".MB_Client_Sending_3.tagsStep."step")
      R_Coil( "MB_TCP_CLIENT".MB_Client_Sending_3.Input.req )
   END_RUNG
   // the same network as SCL:
   #_w1 := ("MB_TCP_CLIENT".MB_Client_Sending_3.tagsStep."step" = 5) AND "MB_TCP_CLIENT".MB_Client_Sending_3.Input.InOut.error;
   IF #_w1 THEN
       "MB_TCP_CLIENT".MB_Client_Sending_3.tagsStep."step" := 1;
       "MB_TCP_CLIENT".MB_Client_Sending_3.Input.req := FALSE;
   END_IF;
END_REGION

REGION Network 14
   // Inicjacja przesłania drugiej części parametrów
   RUNG wire#powerrail
      { S7_Templates := "SrcType := USInt" } EQ_Contact(in1 := "MB_TCP_CLIENT".MB_Client_Sending_3.tagsStep."step", in2 := 6)
      wire#w1
      R_Coil( "MB_TCP_CLIENT".MB_Client_Sending_3.Input.disconnect )
   END_RUNG
   RUNG wire#w1
      I_Contact( "MB_TCP_CLIENT".MB_Client_Sending_3.Input.disconnect )
      Move(in := 7, out1 => "MB_TCP_CLIENT".MB_Client_Sending_3.tagsStep."step")
   END_RUNG
   // the same network as SCL:
   #_w1 := "MB_TCP_CLIENT".MB_Client_Sending_3.tagsStep."step" = 6;
   IF #_w1 THEN "MB_TCP_CLIENT".MB_Client_Sending_3.Input.disconnect := FALSE; END_IF;
   IF #_w1 AND NOT "MB_TCP_CLIENT".MB_Client_Sending_3.Input.disconnect THEN
       "MB_TCP_CLIENT".MB_Client_Sending_3.tagsStep."step" := 7;
   END_IF;
END_REGION

REGION Network 16
   // - wysyłanie do PLC Pompownia
   RUNG wire#powerrail
      { S7_Templates := "SrcType := USInt" } EQ_Contact(in1 := "MB_TCP_CLIENT".MB_Client_Sending_3.tagsStep."step", in2 := 7)
      wire#w1
      { S7_GenerateENO := "TRUE" } Move(in := 502, out1 => "MB_TCP_CLIENT".MB_Client_Sending_3.Input.PORT)
      { S7_GenerateENO := "TRUE" } Move(in := 1, out1 => "MB_TCP_CLIENT".MB_Client_Sending_3.Input.CONNECT_ID)
      { S7_GenerateENO := "TRUE" } Move(in := 1, out1 => "MB_TCP_CLIENT".MB_Client_Sending_3.Input.MB_MODE)
      { S7_GenerateENO := "TRUE" } Move(in := 40034, out1 => "MB_TCP_CLIENT".MB_Client_Sending_3.Input.MB_DATA_ADDR)
      { S7_GenerateENO := "TRUE" } Move(in := 9, out1 => "MB_TCP_CLIENT".MB_Client_Sending_3.Input.DATA_LEN)
      S_Coil( "MB_TCP_CLIENT".MB_Client_Sending_3.Input.req )
   END_RUNG
   RUNG wire#w1
      { S7_GenerateENO := "TRUE" } Move(in := 8, out1 => "MB_TCP_CLIENT".MB_Client_Sending_3.tagsStep."step")
   END_RUNG
   // the same network as SCL:
   // ENO of a box is taken as its EN; it also drops when the box reports an error
   IF "MB_TCP_CLIENT".MB_Client_Sending_3.tagsStep."step" = 7 THEN
       "MB_TCP_CLIENT".MB_Client_Sending_3.Input.PORT := 502;
       "MB_TCP_CLIENT".MB_Client_Sending_3.Input.CONNECT_ID := 1;
       "MB_TCP_CLIENT".MB_Client_Sending_3.Input.MB_MODE := 1;
       "MB_TCP_CLIENT".MB_Client_Sending_3.Input.MB_DATA_ADDR := 40034;
       "MB_TCP_CLIENT".MB_Client_Sending_3.Input.DATA_LEN := 9;
       "MB_TCP_CLIENT".MB_Client_Sending_3.Input.req := TRUE;
       "MB_TCP_CLIENT".MB_Client_Sending_3.tagsStep."step" := 8;
   END_IF;
END_REGION

REGION Network 17: Wysyłanie danych - step 2
   // Analogi
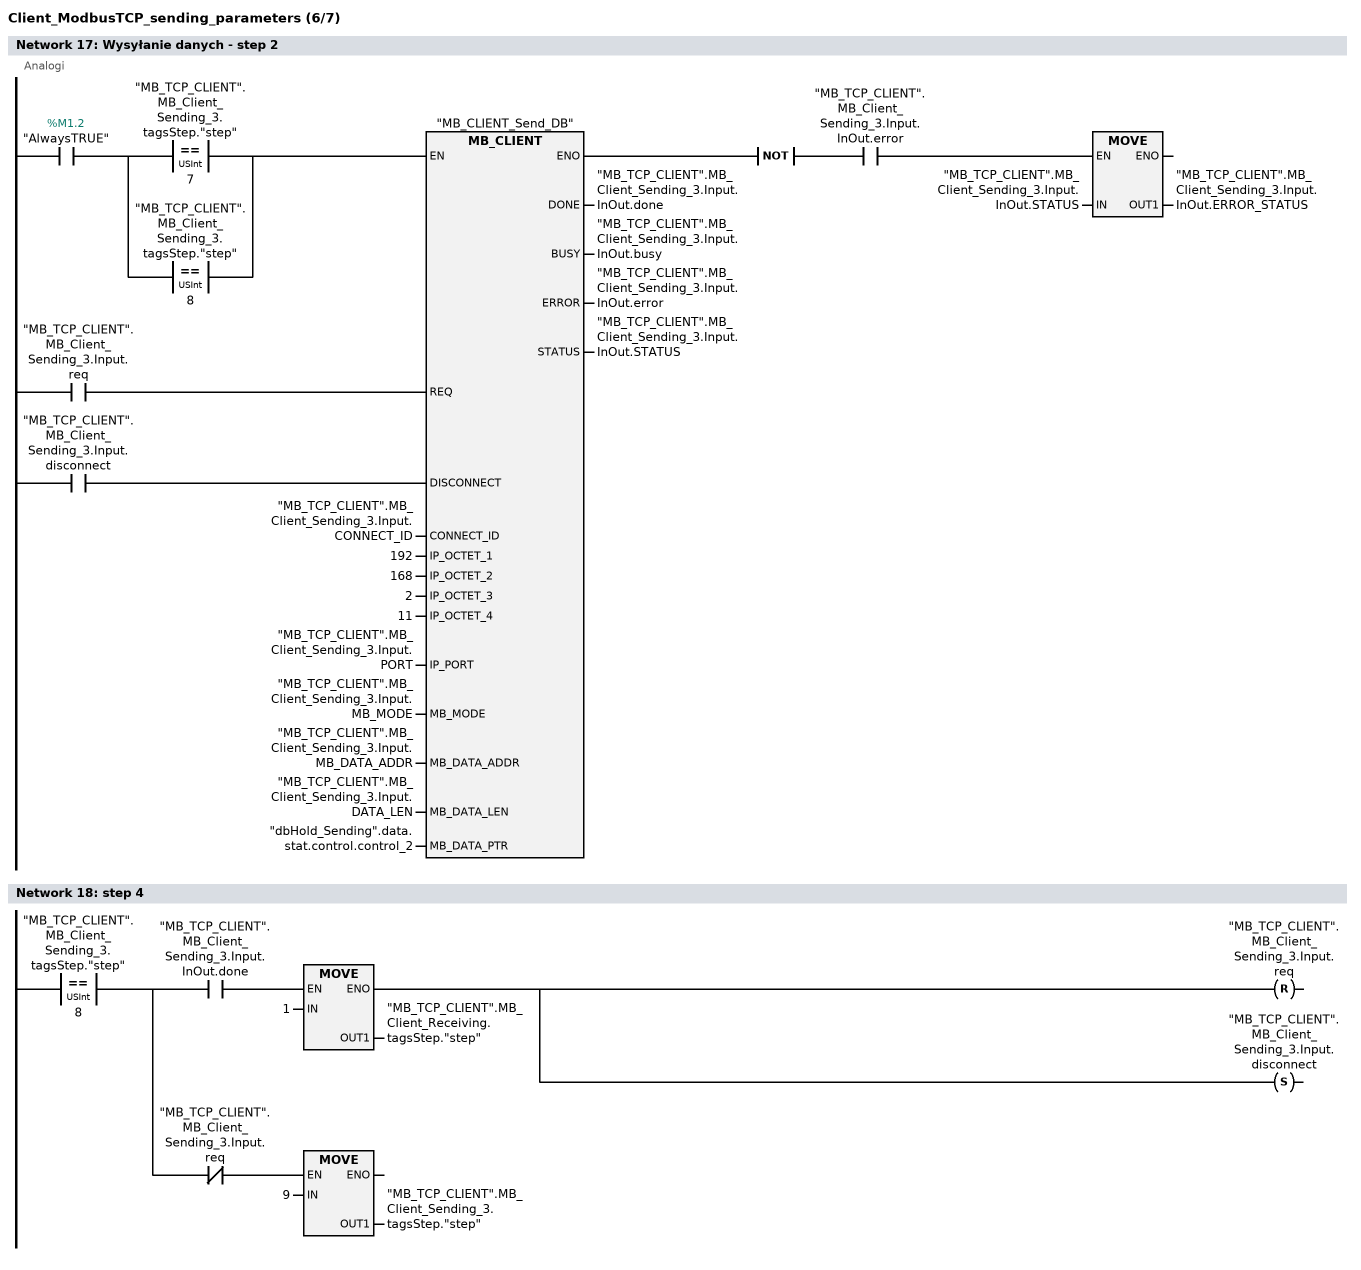
   RUNG wire#powerrail
      Contact( "AlwaysTRUE" )
      wire#w1
      { S7_Templates := "SrcType := USInt" } EQ_Contact(in1 := "MB_TCP_CLIENT".MB_Client_Sending_3.tagsStep."step", in2 := 7)
      wire#w2
      { S7_Templates := "[card1200 := 1, card1500 := 0]" } "MB_CLIENT_Send_DB".MB_CLIENT(REQ := wire#w3, DISCONNECT := wire#w4, CONNECT_ID := "MB_TCP_CLIENT".MB_Client_Sending_3.Input.CONNECT_ID, IP_OCTET_1 := 192, IP_OCTET_2 := 168, IP_OCTET_3 := 2, IP_OCTET_4 := 11, IP_PORT := "MB_TCP_CLIENT".MB_Client_Sending_3.Input.PORT, MB_MODE := "MB_TCP_CLIENT".MB_Client_Sending_3.Input.MB_MODE, MB_DATA_ADDR := "MB_TCP_CLIENT".MB_Client_Sending_3.Input.MB_DATA_ADDR, MB_DATA_LEN := "MB_TCP_CLIENT".MB_Client_Sending_3.Input.DATA_LEN, MB_DATA_PTR := "dbHold_Sending".data.stat.control.control_2, DONE => "MB_TCP_CLIENT".MB_Client_Sending_3.Input.InOut.done, BUSY => "MB_TCP_CLIENT".MB_Client_Sending_3.Input.InOut.busy, ERROR => "MB_TCP_CLIENT".MB_Client_Sending_3.Input.InOut.error, STATUS => "MB_TCP_CLIENT".MB_Client_Sending_3.Input.InOut.STATUS)
      Not()
      Contact( "MB_TCP_CLIENT".MB_Client_Sending_3.Input.InOut.error )
      Move(in := "MB_TCP_CLIENT".MB_Client_Sending_3.Input.InOut.STATUS, out1 => "MB_TCP_CLIENT".MB_Client_Sending_3.Input.InOut.ERROR_STATUS)
   END_RUNG
   RUNG wire#w1
      { S7_Templates := "SrcType := USInt" } EQ_Contact(in1 := "MB_TCP_CLIENT".MB_Client_Sending_3.tagsStep."step", in2 := 8)
   END_RUNG wire#w2
   RUNG wire#powerrail
      Contact( "MB_TCP_CLIENT".MB_Client_Sending_3.Input.req )
   END_RUNG wire#w3
   RUNG wire#powerrail
      Contact( "MB_TCP_CLIENT".MB_Client_Sending_3.Input.disconnect )
   END_RUNG wire#w4
   // the same network as SCL:
   #_w1 := "AlwaysTRUE" AND (("MB_TCP_CLIENT".MB_Client_Sending_3.tagsStep."step" = 7) OR ("MB_TCP_CLIENT".MB_Client_Sending_3.tagsStep."step" = 8));
   "MB_CLIENT_Send_DB"(EN := #_w1,   // MB_CLIENT
                       REQ := "MB_TCP_CLIENT".MB_Client_Sending_3.Input.req,
                       DISCONNECT := "MB_TCP_CLIENT".MB_Client_Sending_3.Input.disconnect,
                       CONNECT_ID := "MB_TCP_CLIENT".MB_Client_Sending_3.Input.CONNECT_ID,
                       IP_OCTET_1 := 192,
                       IP_OCTET_2 := 168,
                       IP_OCTET_3 := 2,
                       IP_OCTET_4 := 11,
                       IP_PORT := "MB_TCP_CLIENT".MB_Client_Sending_3.Input.PORT,
                       MB_MODE := "MB_TCP_CLIENT".MB_Client_Sending_3.Input.MB_MODE,
                       MB_DATA_ADDR := "MB_TCP_CLIENT".MB_Client_Sending_3.Input.MB_DATA_ADDR,
                       MB_DATA_LEN := "MB_TCP_CLIENT".MB_Client_Sending_3.Input.DATA_LEN,
                       MB_DATA_PTR := "dbHold_Sending".data.stat.control.control_2,
                       DONE => "MB_TCP_CLIENT".MB_Client_Sending_3.Input.InOut.done,
                       BUSY => "MB_TCP_CLIENT".MB_Client_Sending_3.Input.InOut.busy,
                       ERROR => "MB_TCP_CLIENT".MB_Client_Sending_3.Input.InOut.error,
                       STATUS => "MB_TCP_CLIENT".MB_Client_Sending_3.Input.InOut.STATUS,
                       ENO => #_w2);
   IF NOT #_w2 AND "MB_TCP_CLIENT".MB_Client_Sending_3.Input.InOut.error THEN
       "MB_TCP_CLIENT".MB_Client_Sending_3.Input.InOut.ERROR_STATUS := "MB_TCP_CLIENT".MB_Client_Sending_3.Input.InOut.STATUS;
   END_IF;
END_REGION

REGION Network 18: step 4
   RUNG wire#powerrail
      { S7_Templates := "SrcType := USInt" } EQ_Contact(in1 := "MB_TCP_CLIENT".MB_Client_Sending_3.tagsStep."step", in2 := 8)
      wire#w1
      Contact( "MB_TCP_CLIENT".MB_Client_Sending_3.Input.InOut.done )
      Move(in := 1, out1 => "MB_TCP_CLIENT".MB_Client_Receiving.tagsStep."step")
      wire#w2
      R_Coil( "MB_TCP_CLIENT".MB_Client_Sending_3.Input.req )
   END_RUNG
   RUNG wire#w2
      S_Coil( "MB_TCP_CLIENT".MB_Client_Sending_3.Input.disconnect )
   END_RUNG
   RUNG wire#w1
      I_Contact( "MB_TCP_CLIENT".MB_Client_Sending_3.Input.req )
      Move(in := 9, out1 => "MB_TCP_CLIENT".MB_Client_Sending_3.tagsStep."step")
   END_RUNG
   // the same network as SCL:
   #_w1 := "MB_TCP_CLIENT".MB_Client_Sending_3.tagsStep."step" = 8;
   IF #_w1 AND "MB_TCP_CLIENT".MB_Client_Sending_3.Input.InOut.done THEN
       "MB_TCP_CLIENT".MB_Client_Receiving.tagsStep."step" := 1;
       "MB_TCP_CLIENT".MB_Client_Sending_3.Input.req := FALSE;
       "MB_TCP_CLIENT".MB_Client_Sending_3.Input.disconnect := TRUE;
   END_IF;
   IF #_w1 AND NOT "MB_TCP_CLIENT".MB_Client_Sending_3.Input.req THEN
       "MB_TCP_CLIENT".MB_Client_Sending_3.tagsStep."step" := 9;
   END_IF;
END_REGION

REGION Network 19
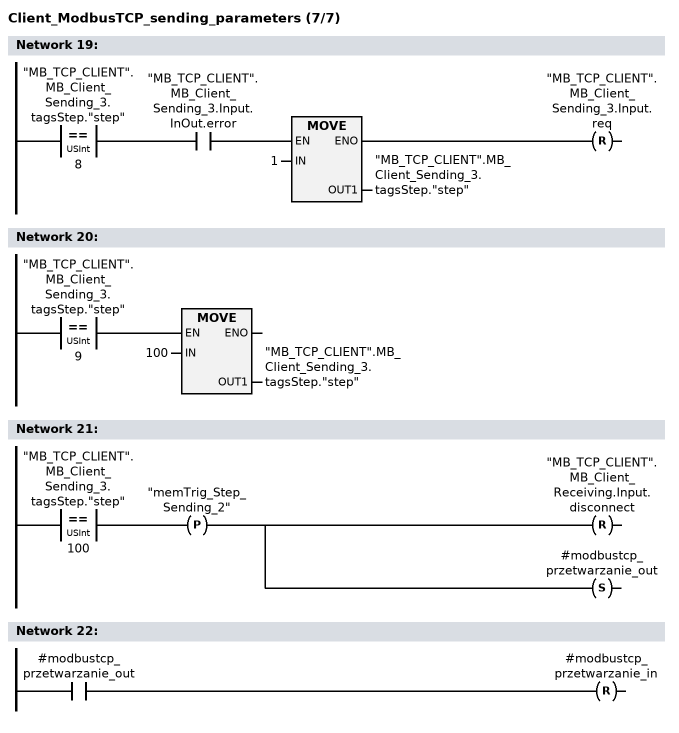
   RUNG wire#powerrail
      { S7_Templates := "SrcType := USInt" } EQ_Contact(in1 := "MB_TCP_CLIENT".MB_Client_Sending_3.tagsStep."step", in2 := 8)
      Contact( "MB_TCP_CLIENT".MB_Client_Sending_3.Input.InOut.error )
      Move(in := 1, out1 => "MB_TCP_CLIENT".MB_Client_Sending_3.tagsStep."step")
      R_Coil( "MB_TCP_CLIENT".MB_Client_Sending_3.Input.req )
   END_RUNG
   // the same network as SCL:
   #_w1 := ("MB_TCP_CLIENT".MB_Client_Sending_3.tagsStep."step" = 8) AND "MB_TCP_CLIENT".MB_Client_Sending_3.Input.InOut.error;
   IF #_w1 THEN
       "MB_TCP_CLIENT".MB_Client_Sending_3.tagsStep."step" := 1;
       "MB_TCP_CLIENT".MB_Client_Sending_3.Input.req := FALSE;
   END_IF;
END_REGION

REGION Network 20
   RUNG wire#powerrail
      { S7_Templates := "SrcType := USInt" } EQ_Contact(in1 := "MB_TCP_CLIENT".MB_Client_Sending_3.tagsStep."step", in2 := 9)
      Move(in := 100, out1 => "MB_TCP_CLIENT".MB_Client_Sending_3.tagsStep."step")
   END_RUNG
   // the same network as SCL:
   IF "MB_TCP_CLIENT".MB_Client_Sending_3.tagsStep."step" = 9 THEN
       "MB_TCP_CLIENT".MB_Client_Sending_3.tagsStep."step" := 100;
   END_IF;
END_REGION

REGION Network 21
   RUNG wire#powerrail
      { S7_Templates := "SrcType := USInt" } EQ_Contact(in1 := "MB_TCP_CLIENT".MB_Client_Sending_3.tagsStep."step", in2 := 100)
      P_Trig( "memTrig_Step_Sending_2" )
      wire#w1
      R_Coil( "MB_TCP_CLIENT".MB_Client_Receiving.Input.disconnect )
   END_RUNG
   RUNG wire#w1
      S_Coil( #modbustcp_przetwarzanie_out )
   END_RUNG
   // the same network as SCL:
   #_w1 := "MB_TCP_CLIENT".MB_Client_Sending_3.tagsStep."step" = 100;
   #_w2 := #_w1 AND NOT "memTrig_Step_Sending_2";   // rising edge
   "memTrig_Step_Sending_2" := #_w1;
   IF #_w2 THEN
       "MB_TCP_CLIENT".MB_Client_Receiving.Input.disconnect := FALSE;
       #modbustcp_przetwarzanie_out := TRUE;
   END_IF;
END_REGION

REGION Network 22
   RUNG wire#powerrail
      Contact( #modbustcp_przetwarzanie_out )
      R_Coil( #modbustcp_przetwarzanie_in )
   END_RUNG
   // the same network as SCL:
   IF #modbustcp_przetwarzanie_out THEN #modbustcp_przetwarzanie_in := FALSE; END_IF;
END_REGION
END_FUNCTION_BLOCK

FUNCTION "clear-drive_error" : Void
TITLE = kasowanie alarmów
{ S7_Optimized_Access := 'TRUE' }
AUTHOR : rtecmer
VERSION : 0.1
//Funkcja kasowania alarmów napedów. Kasowanie zdalne z MT101 poprzez SCADA. MT101 komunikuje się poprzez modbus rtu przeniesienie wartości do semdin modbus tcp i przetworzenie sygnału sterowania

BEGIN
	(*
	//=============================================================================
	//(JZWiK S.A Radosław Tecmer)
	//(c)Copyright (2021) All Rights Reserved
	//-----------------------------------------------------------------------------
	//Testowane z:   (system docelowy z  FW 4.2)
	//Pakiet inżynierski:   TIA Portal (V14 Sp1 Update 9)
	//Ograniczenia:  ( - )
	//Wymagania:  (minimalne S7-1200 CPU 1214 FW 3.2 .)
	//Funkcjonalnośc: (Pzetwarzanie sygnałów z MT101 protokołem Modbus RTU - TCP. 
	                    Kasowanie alarów)
	//-----------------------------------------------------------------------------
	//Zmainy wprowadzone:
	//Wersja  Data       Osoba wprowadzająca zmiany - ekspert
	//01.00.00 17.11.2021 (Tecmer Radosław - twórca) Pieresza wersja 01.00.00
	//=============================================================================
	*)
	
	REGION Z1
	  // 
	  //Ustawienie bitu Reset dla Drive Motor Z1
	  %DB10.DBX6.6 := %DB58.DBX19.4;
	  IF %DB10.DBX6.0 = FALSE AND %DB58.DBX19.4 = TRUE THEN
	    //Ustawienie w automat 
	    %DB10.DBX6.7 := TRUE;
	    // Kasowanie bitu RESET Driver i Modbus bit Reset
	    %DB10.DBX6.0 := FALSE;
	    %DB58.DBX19.4 := False;
	    ;
	  END_IF;
	  
	  
	END_REGION
	
	REGION Z2
	  // 
	  //Ustawienie bitu Reset dla Drive Motor Z2
	  %DB10.DBX8.6 := %DB58.DBX19.5;
	  IF %DB10.DBX8.0 = FALSE AND %DB58.DBX19.5 = TRUE THEN
	    //Ustawienie w automat 
	    %DB10.DBX8.7 := TRUE;
	    // Kasowanie bitu RESET Driver i Modbus bit Reset
	    %DB10.DBX8.0 := FALSE;
	    %DB58.DBX19.5 := False;
	    ;
	  END_IF;
	  
	  
	END_REGION
	
	REGION Z3
	  // 
	  //Ustawienie bitu Reset dla Drive Motor Z3
	  %DB10.DBX10.6 := %DB58.DBX19.6;
	  IF %DB10.DBX10.0 = FALSE AND %DB58.DBX19.6 = TRUE THEN
	    //Ustawienie w automat 
	    %DB10.DBX10.7 := TRUE;
	    // Kasowanie bitu RESET Driver i Modbus bit Reset
	    %DB10.DBX10.0 := FALSE;
	    %DB58.DBX19.6 := False;
	    ;
	  END_IF;
	  
	  
	END_REGION
	
	REGION Z4
	  // 
	  //Ustawienie bitu Reset dla Drive Motor Z4
	  %DB10.DBX12.6 := %DB58.DBX19.7;
	  IF %DB10.DBX12.0 = FALSE AND %DB58.DBX19.7 = TRUE THEN
	    //Ustawienie w automat 
	    %DB10.DBX12.7 := TRUE;
	    // Kasowanie bitu RESET Driver i Modbus bit Reset
	    %DB10.DBX12.0 := FALSE;
	    %DB58.DBX19.7 := False;
	    ;
	  END_IF;
	  
	  
	END_REGION
	
	REGION Z5
	  // 
	  //Ustawienie bitu Reset dla Drive Motor Z5
	  %DB10.DBX14.6 := %DB58.DBX18.0;
	  IF %DB10.DBX14.0 = FALSE AND %DB58.DBX18.0 = TRUE THEN
	    //Ustawienie w automat 
	    %DB10.DBX14.7 := TRUE;
	    // Kasowanie bitu RESET Driver i Modbus bit Reset
	    %DB10.DBX14.0 := FALSE;
	    %DB58.DBX18.0 := False;
	    ;
	  END_IF;
	  
	  
	END_REGION
	
	REGION Z6
	  // 
	  //Ustawienie bitu Reset dla Drive Motor Z6
	  %DB10.DBX16.6 := %DB58.DBX18.1;
	  IF %DB10.DBX16.0 = FALSE AND %DB58.DBX18.1 = TRUE THEN
	    //Ustawienie w automat 
	    %DB10.DBX16.7 := TRUE;
	    // Kasowanie bitu RESET Driver i Modbus bit Reset
	    %DB10.DBX16.0 := FALSE;
	    %DB58.DBX18.1 := False;
	    ;
	  END_IF;
	  
	  
	END_REGION
	
	REGION Z7
	  // 
	  //Ustawienie bitu Reset dla Drive Motor Z7
	  %DB10.DBX18.6 := %DB58.DBX18.2;
	  IF %DB10.DBX18.0 = FALSE AND %DB58.DBX18.2 = TRUE THEN
	    //Ustawienie w automat 
	    %DB10.DBX18.7 := TRUE;
	    // Kasowanie bitu RESET Driver i Modbus bit Reset
	    %DB10.DBX18.0 := FALSE;
	    %DB58.DBX18.2 := False;
	    ;
	  END_IF;
	  
	  
	END_REGION
	
	REGION Z8
	  // 
	  //Ustawienie bitu Reset dla Drive Motor Z8
	  %DB10.DBX20.6 := %DB58.DBX18.3;
	  IF %DB10.DBX20.0 = FALSE AND %DB58.DBX18.3 = TRUE THEN
	    //Ustawienie w automat 
	    %DB10.DBX20.7 := TRUE;
	    // Kasowanie bitu RESET Driver i Modbus bit Reset
	    %DB10.DBX20.0 := FALSE;
	    %DB58.DBX18.3 := False;
	    ;
	  END_IF;
	  
	  
	END_REGION
	
	REGION Z9
	  // 
	  //Ustawienie bitu Reset dla Drive Motor Z9
	  %DB10.DBX22.6 := %DB58.DBX18.4;
	  IF %DB10.DBX22.0 = FALSE AND %DB58.DBX18.4 = TRUE THEN
	    //Ustawienie w automat 
	    %DB10.DBX22.7 := TRUE;
	    // Kasowanie bitu RESET Driver i Modbus bit Reset
	    %DB10.DBX22.0 := FALSE;
	    %DB58.DBX18.4 := False;
	    ;
	  END_IF;
	  
	  
	END_REGION
	
	REGION Z10
	  // 
	  //Ustawienie bitu Reset dla Drive Motor Z10
	  %DB10.DBX24.6 := %DB58.DBX18.5;
	  IF %DB10.DBX24.0 = FALSE AND %DB58.DBX18.5 = TRUE THEN
	    //Ustawienie w automat 
	    %DB10.DBX24.7 := TRUE;
	    // Kasowanie bitu RESET Driver i Modbus bit Reset
	    %DB10.DBX24.0 := FALSE;
	    %DB58.DBX18.5 := False;
	    ;
	  END_IF;
	  
	  
	END_REGION
	
	
	
	
	
	
	
	
	
	
	
	
END_FUNCTION

FUNCTION_BLOCK "operating_mode_select_aut-man"
TITLE = Przełącznik Trybu Pracy Napędów
{ S7_Optimized_Access := 'TRUE' }
AUTHOR : rtecmer
VERSION : 0.1
//Funkcja przeprowadza sptawdzenie stanu zmiany sygnału  na zmiennych wyboru trybu pracy napeów i jesli strwierdzi zmianę stanu zmennej to wykonuje zmianę trybu na AUT
   VAR 
      setTrig_Z1 : Bool;   // bit pomocniczy przełączenia trybu
      setTrig_Z2 : Bool := false;   // bit pomocniczy przełączenia trybu
      setTrig_Z3 : Bool := false;   // bit pomocniczy przełączenia trybu
      setTrig_Z4 : Bool := false;   // bit pomocniczy przełączenia trybu
      setTrig_Z5 : Bool := false;   // bit pomocniczy przełączenia trybu
      setTrig_Z6 : Bool := false;   // bit pomocniczy przełączenia trybu
      setTrig_Z7 : Bool := false;   // bit pomocniczy przełączenia trybu
      setTrig_Z8 : Bool := false;   // bit pomocniczy przełączenia trybu
      setTrig_Z9 : Bool := false;   // bit pomocniczy przełączenia trybu
      setTrig_Z10 : Bool := false;   // bit pomocniczy przełączenia trybu
      set_aut_man_Z1 : Bool;   // bit pomocniczy sterowania trybem
      set_aut_man_Z2 : Bool := false;   // bit pomocniczy sterowania trybem
      set_aut_man_Z3 : Bool := false;   // bit pomocniczy sterowania trybem
      set_aut_man_Z4 : Bool := false;   // bit pomocniczy sterowania trybem
      set_aut_man_Z5 : Bool := false;   // bit pomocniczy sterowania trybem
      set_aut_man_Z6 : Bool := false;   // bit pomocniczy sterowania trybem
      set_aut_man_Z7 : Bool := false;   // bit pomocniczy sterowania trybem
      set_aut_man_Z8 : Bool := false;   // bit pomocniczy sterowania trybem
      set_aut_man_Z9 : Bool := false;   // bit pomocniczy sterowania trybem
      set_aut_man_Z10 : Bool := false;   // bit pomocniczy sterowania trybem
   END_VAR


BEGIN
	(*
	//=============================================================================
	//(JZWiK S.A Radosław Tecmer)
	//(c)Copyright (2021) All Rights Reserved
	//-----------------------------------------------------------------------------
	//Testowane z:   (system docelowy z  FW 4.2)
	//Pakiet inżynierski:   TIA Portal (V14 Sp1 Update 9)
	//Ograniczenia:  ( - )
	//Wymagania:  (minimalne S7-1200 CPU 1214 FW 3.2 .)
	//Funkcjonalnośc: (Pzetwarzanie sygnałów z MT101 protokołem Modbus RTU. 
	                    Wybór Trybu Pracy Napędu)
	//-----------------------------------------------------------------------------
	//Zmainy wprowadzone:
	//Wersja  Data       Osoba wprowadzająca zmiany - ekspert
	//01.00.00 17.06.2022 (Tecmer Radosław - twórca) Pieresza wersja 01.00.00
	//=============================================================================
	*)
	
	//--- Wybór Trybu Pracy Aut/Man Sterowanie Otwórz/ Zamknij
	
	REGION //Drive Motor Z1 ustaw na  Automat/Manual/Otwarta/Zamknięta
	  IF %DB58.DBX14.0 OR %DB58.DBX17.4 THEN
	    // przełączniki bistabilny każdy stan Hi powoduje zmianę przełącznika 
	    #set_aut_man_Z1 := TRUE;
	  ELSE
	    #set_aut_man_Z1 := FALSE;
	    ;
	  END_IF;
	  
	  IF %DB10.DBX6.0 = FALSE THEN
	    // przełącznik bistabilny
	    "R_TRIG_DB_AUT_Z1"(CLK := #set_aut_man_Z1,
	                       Q => #setTrig_Z1);
	    ;
	  END_IF;
	  // przełącz na automat
	  IF #setTrig_Z1 = TRUE AND %DB58.DBX14.0 = TRUE THEN
	    %DB10.DBX6.7 := TRUE;
	    ;
	  END_IF;
	  //przełącz na manual
	  IF #setTrig_Z1 = TRUE AND %DB58.DBX17.4 = TRUE THEN
	    %DB10.DBX6.7 := FALSE;
	    ;
	  END_IF;
	  
	  IF (%DB10.DBX7.7 = TRUE AND %DB58.DBX14.0 = TRUE) OR (%DB10.DBX7.7 = FALSE AND %DB58.DBX17.4 = TRUE) THEN
	    // Wyczyść całą zmienną
	    "dbHoldRegSlave_to_MT101".Status_Sterowanie.instConrol_ManAut_1 := 0;
	    "dbHold_Sending".data.stat.control.control_2.set_res_bity_tryb_napędów_1 := 0;
	    "dbHoldRegSlave_to_MT101".Status_Sterowanie.instConrol_ManAut_2 := 0;
	    "dbHold_Sending".data.stat.control.control_2.set_res_bity_tryb_napędów_2 := 0;
	    %DB58.DBX14.0 := FALSE;
	    %DB58.DBX17.4:= FALSE
	    ;
	  END_IF;
	  
	  // sterowanie OTWIERANIE - ZAMYKANIE
	  // Otwórz/
	  // przekazanie bitu roskazu z bloku modbus rtu do bloku statusu napędu
	  %DB10.DBX6.4 := %DB58.DBX10.0; //ustawienie bitu otwieranie
	  IF %DB58.DBX10.0 AND %DB10.DBX7.1 THEN
	    //jeśli ustawiony bit otwierania z modbus i potwierdzone otwarcie 
	    %DB58.DBX10.0 := FALSE; // kasuj bit roskazu
	    "dbHoldRegSlave_to_MT101".Status_Sterowanie.instControllDrivers_1 := 0;
	 
	    "dbHoldRegSlave_to_MT101".Status_Sterowanie.instControllDrivers_2 := 0;
	   
	   
	    ;
	  END_IF;
	  //Zamknij
	  //przekazanie bitu roskazu z bloku modbus rtu do bloku statusu napędu
	  %DB10.DBX6.5 := %DB58.DBX13.4; //ustawienie bitu zamykanie
	  IF %DB58.DBX13.4 AND %DB10.DBX7.3 = FALSE THEN
	    //jeśli ustawiony bit zamykanie z modbus i potwierdzone zamknięcie 
	    %DB58.DBX13.4 := FALSE; // kasuj bit roskazu
	    "dbHoldRegSlave_to_MT101".Status_Sterowanie.instControllDrivers_1 := 0;
	
	    "dbHoldRegSlave_to_MT101".Status_Sterowanie.instControllDrivers_2 := 0;
	    
	    ;
	  END_IF;
	  
	END_REGION
	
	
	REGION //Drive Motor Z2 ustaw na  Automat/Manual/Otwarta/Zamknięta
	  IF %DB58.DBX14.1 OR %DB58.DBX17.5 THEN
	    //przełączniki bistabilny każdy stan Hi powoduje zmianę przełącznika  
	    #set_aut_man_Z2 := TRUE;
	  ELSE
	    #set_aut_man_Z2 := FALSE;
	    ;
	  END_IF;
	  
	  IF %DB10.DBX8.0 = FALSE THEN
	    //przełącznik bistabilny
	    "R_TRIG_DB_AUT_Z2"(CLK :=#set_aut_man_Z2,
	                       Q => #setTrig_Z2);
	    ;
	  END_IF;
	  // przełącz na automat
	  IF #setTrig_Z2 = TRUE AND %DB58.DBX14.1 = TRUE THEN
	    %DB10.DBX8.7 := TRUE;
	    ;
	  END_IF;
	  //przełącz na manual
	  IF #setTrig_Z2 = TRUE AND %DB58.DBX17.5 = TRUE THEN
	    %DB10.DBX8.7 := FALSE;
	    ;
	  END_IF;
	  
	  IF (%DB10.DBX9.7 = TRUE AND %DB58.DBX14.1 = TRUE) OR (%DB10.DBX9.7 = FALSE AND %DB58.DBX17.5 = TRUE) THEN
	    // Wyczyść całą zmienną
	    "dbHoldRegSlave_to_MT101".Status_Sterowanie.instConrol_ManAut_1 := 0;
	    "dbHold_Sending".data.stat.control.control_2.set_res_bity_tryb_napędów_1 := 0;
	    "dbHoldRegSlave_to_MT101".Status_Sterowanie.instConrol_ManAut_2 := 0;
	    "dbHold_Sending".data.stat.control.control_2.set_res_bity_tryb_napędów_2 := 0;
	    %DB58.DBX14.1 := FALSE;
	    %DB58.DBX17.5 := FALSE;
	    ;
	  END_IF;
	  
	  // sterowanie OTWIERANIE - ZAMYKANIE
	  // Otwórz/
	  // przekazanie bitu roskazu z bloku modbus rtu do bloku statusu napędu
	  %DB10.DBX8.4 := %DB58.DBX10.1; //ustawienie bitu otwieranie
	  IF %DB58.DBX10.1 AND %DB10.DBX9.1 THEN
	    //jeśli ustawiony bit otwierania z modbus i potwierdzone otwarcie 
	    %DB58.DBX10.1 := FALSE; // kasuj bit roskazu
	    "dbHoldRegSlave_to_MT101".Status_Sterowanie.instControllDrivers_1 := 0;
	    
	    "dbHoldRegSlave_to_MT101".Status_Sterowanie.instControllDrivers_2 := 0;
	    
	    
	    ;
	  END_IF;
	  //Zamknij
	  //przekazanie bitu roskazu z bloku modbus rtu do bloku statusu napędu
	  %DB10.DBX8.5 := %DB58.DBX13.5; //ustawienie bitu zamykanie
	  IF %DB58.DBX13.5 AND %DB10.DBX9.3 = FALSE THEN
	    //jeśli ustawiony bit zamykanie z modbus i potwierdzone zamknięcie 
	    %DB58.DBX13.5 := FALSE; // kasuj bit roskazu
	    "dbHoldRegSlave_to_MT101".Status_Sterowanie.instControllDrivers_1 := 0;
	    
	    "dbHoldRegSlave_to_MT101".Status_Sterowanie.instControllDrivers_2 := 0;
	    
	    ;
	  END_IF;
	  
	  
	END_REGION
	
	
	REGION //Drive Motor Z3 ustaw na  Automat/Manual/Otwarta/Zamknięta
	  IF %DB58.DBX14.2 OR %DB58.DBX17.6 THEN
	    //przełączniki bistabilny każdy stan Hi powoduje zmianę przełącznika  
	    #set_aut_man_Z3 := TRUE;
	  ELSE
	    #set_aut_man_Z3 := FALSE
	    ;
	  END_IF;
	  
	  IF %DB10.DBX10.0 = FALSE THEN
	    // przełącznik bistabilny
	    "R_TRIG_DB_AUT_Z3"(CLK := #set_aut_man_Z3,
	                       Q => #setTrig_Z3);
	    ;
	  END_IF;
	  // przełącz na automat
	  IF #setTrig_Z3 = TRUE AND %DB58.DBX14.2 = TRUE THEN
	    %DB10.DBX10.7 := TRUE;
	    ;
	  END_IF;
	  //przełącz na manual
	  IF #setTrig_Z3 = TRUE AND %DB58.DBX17.6 = TRUE THEN
	    %DB10.DBX10.7 := FALSE;
	    ;
	  END_IF;
	  
	  IF (%DB10.DBX11.7 = TRUE AND %DB58.DBX14.2) OR (%DB10.DBX11.7 = FALSE AND %DB58.DBX17.6) THEN
	    // Wyczyść całą zmienną
	    "dbHoldRegSlave_to_MT101".Status_Sterowanie.instConrol_ManAut_1 := 0;
	    "dbHold_Sending".data.stat.control.control_2.set_res_bity_tryb_napędów_1 := 0;
	    "dbHoldRegSlave_to_MT101".Status_Sterowanie.instConrol_ManAut_2 := 0;
	    "dbHold_Sending".data.stat.control.control_2.set_res_bity_tryb_napędów_2 := 0;
	    %DB58.DBX14.2 := FALSE;
	    %DB58.DBX17.6 := FALSE
	    ;
	  END_IF;
	  
	  // sterowanie OTWIERANIE - ZAMYKANIE
	  // Otwórz/
	  // przekazanie bitu roskazu z bloku modbus rtu do bloku statusu napędu
	  %DB10.DBX10.4 := %DB58.DBX10.2; //ustawienie bitu otwieranie
	  IF %DB58.DBX10.2 AND %DB10.DBX11.1 THEN
	    //jeśli ustawiony bit otwierania z modbus i potwierdzone otwarcie 
	    %DB58.DBX10.2 := FALSE; // kasuj bit roskazu
	    "dbHoldRegSlave_to_MT101".Status_Sterowanie.instControllDrivers_1 := 0;
	    
	    "dbHoldRegSlave_to_MT101".Status_Sterowanie.instControllDrivers_2 := 0;
	    
	    
	    ;
	  END_IF;
	  //Zamknij
	  //przekazanie bitu roskazu z bloku modbus rtu do bloku statusu napędu
	  %DB10.DBX10.5 := %DB58.DBX13.6; //ustawienie bitu zamykanie
	  IF %DB58.DBX13.6 AND %DB10.DBX11.3 = FALSE THEN
	    //jeśli ustawiony bit zamykanie z modbus i potwierdzone zamknięcie 
	    %DB58.DBX13.6 := FALSE; // kasuj bit roskazu
	    "dbHoldRegSlave_to_MT101".Status_Sterowanie.instControllDrivers_1 := 0;
	    
	    "dbHoldRegSlave_to_MT101".Status_Sterowanie.instControllDrivers_2 := 0;
	    
	    ;
	  END_IF;
	  
	END_REGION
	
	
	REGION //Drive Motor Z4 ustaw na  Automat/Manual/Otwarta/Zamknięta
	  IF %DB58.DBX14.3 OR %DB58.DBX17.7 THEN
	    //przełączniki bistabilny każdy stan Hi powoduje zmianę przełącznika 
	    #set_aut_man_Z4 := TRUE;
	  ELSE
	    #set_aut_man_Z4 := FALSE
	    ;
	  END_IF;
	  
	  IF %DB10.DBX12.0 = FALSE THEN
	    // przełącznik bistabilny
	    "R_TRIG_DB_AUT_Z4"(CLK := #set_aut_man_Z4,
	                       Q => #setTrig_Z4);
	    ;
	  END_IF;
	  
	  IF #setTrig_Z4 = TRUE AND %DB58.DBX14.3 = TRUE THEN
	    %DB10.DBX12.7 := TRUE;
	    ;
	  END_IF;
	  
	  IF #setTrig_Z4 = TRUE AND %DB58.DBX17.7 = TRUE THEN
	    %DB10.DBX12.7 := FALSE;
	    ;
	  END_IF;
	  
	  IF (%DB10.DBX13.7 = TRUE AND %DB58.DBX14.3 = TRUE) OR (%DB10.DBX13.7 = FALSE AND %DB58.DBX17.7 = TRUE) THEN
	    // Wyczyść całą zmienną
	    "dbHoldRegSlave_to_MT101".Status_Sterowanie.instConrol_ManAut_1 := 0;
	    "dbHold_Sending".data.stat.control.control_2.set_res_bity_tryb_napędów_1 := 0;
	    "dbHoldRegSlave_to_MT101".Status_Sterowanie.instConrol_ManAut_2 := 0;
	    "dbHold_Sending".data.stat.control.control_2.set_res_bity_tryb_napędów_2 := 0;
	    %DB58.DBX14.3 := FALSE;
	    %DB58.DBX17.7 := FALSE;
	    ;
	  END_IF;
	  
	  // sterowanie OTWIERANIE - ZAMYKANIE
	  // Otwórz/
	  // przekazanie bitu roskazu z bloku modbus rtu do bloku statusu napędu
	  %DB10.DBX12.4 := %DB58.DBX10.3; //ustawienie bitu otwieranie
	  IF %DB58.DBX10.3 AND %DB10.DBX13.1 THEN
	    //jeśli ustawiony bit otwierania z modbus i potwierdzone otwarcie 
	    %DB58.DBX10.3 := FALSE; // kasuj bit roskazu
	    "dbHoldRegSlave_to_MT101".Status_Sterowanie.instControllDrivers_1 := 0;
	    
	    "dbHoldRegSlave_to_MT101".Status_Sterowanie.instControllDrivers_2 := 0;
	    
	    
	    ;
	  END_IF;
	  //Zamknij
	  //przekazanie bitu roskazu z bloku modbus rtu do bloku statusu napędu
	  %DB10.DBX12.5 := %DB58.DBX13.7; //ustawienie bitu zamykanie
	  IF %DB58.DBX13.7 AND %DB10.DBX13.3 = FALSE THEN
	    //jeśli ustawiony bit zamykanie z modbus i potwierdzone zamknięcie 
	    %DB58.DBX13.7 := FALSE; // kasuj bit roskazu
	    "dbHoldRegSlave_to_MT101".Status_Sterowanie.instControllDrivers_1 := 0;
	    
	    "dbHoldRegSlave_to_MT101".Status_Sterowanie.instControllDrivers_2 := 0;
	    
	    ;
	  END_IF;
	  
	END_REGION
	
	REGION //Drive Motor Z5 ustaw na  Automat/Manual/Otwarta/Zamknięta
	  IF %DB58.DBX14.4 OR %DB58.DBX16.0 THEN
	    // //przełączniki bistabilny każdy stan Hi powoduje zmianę przełącznika 
	    #set_aut_man_Z5 := TRUE;
	  ELSE
	    #set_aut_man_Z5 := FALSE
	    ;
	  END_IF;
	  
	  IF %DB10.DBX14.0 = FALSE THEN
	    // gdy brak awarii
	    "R_TRIG_DB_AUT_Z5"(CLK := #set_aut_man_Z5,
	                       Q => #setTrig_Z5);
	    ;
	  END_IF;
	  // przełącz na automat
	  IF #setTrig_Z5 = TRUE AND %DB58.DBX14.4 THEN
	    %DB10.DBX14.7 := TRUE;
	    ;
	  END_IF;
	  // przełącz na manual
	  IF #setTrig_Z5 = TRUE AND %DB58.DBX16.0 THEN
	    %DB10.DBX14.7 := FALSE;
	    ;
	  END_IF;
	  
	  IF (%DB10.DBX15.7 = TRUE AND %DB58.DBX14.4 = TRUE) OR (%DB10.DBX15.7 = FALSE AND %DB58.DBX16.0 = TRUE) THEN
	    // Wyczyść całą zmienną
	    "dbHoldRegSlave_to_MT101".Status_Sterowanie.instConrol_ManAut_1 := 0;
	    "dbHold_Sending".data.stat.control.control_2.set_res_bity_tryb_napędów_1 := 0;
	    "dbHoldRegSlave_to_MT101".Status_Sterowanie.instConrol_ManAut_2 := 0;
	    "dbHold_Sending".data.stat.control.control_2.set_res_bity_tryb_napędów_2 := 0;
	    %DB58.DBX14.4 := FALSE;
	    %DB58.DBX16.0 := FALSE
	    ;
	  END_IF;
	  
	  // sterowanie OTWIERANIE - ZAMYKANIE
	  // Otwórz/
	  // przekazanie bitu roskazu z bloku modbus rtu do bloku statusu napędu
	  %DB10.DBX14.4 := %DB58.DBX10.4; //ustawienie bitu otwieranie
	  IF %DB58.DBX10.4 AND %DB10.DBX15.1 THEN
	    //jeśli ustawiony bit otwierania z modbus i potwierdzone otwarcie 
	    %DB58.DBX10.4 := FALSE; // kasuj bit roskazu
	    "dbHoldRegSlave_to_MT101".Status_Sterowanie.instControllDrivers_1 := 0;
	    
	    "dbHoldRegSlave_to_MT101".Status_Sterowanie.instControllDrivers_2 := 0;
	    
	    
	    ;
	  END_IF;
	  //Zamknij
	  //przekazanie bitu roskazu z bloku modbus rtu do bloku statusu napędu
	  %DB10.DBX14.5 := %DB58.DBX12.0; //ustawienie bitu zamykanie
	  IF %DB58.DBX12.0 AND %DB10.DBX15.3 = FALSE THEN
	    //jeśli ustawiony bit zamykanie z modbus i potwierdzone zamknięcie 
	    %DB58.DBX12.0 := FALSE; // kasuj bit roskazu
	    "dbHoldRegSlave_to_MT101".Status_Sterowanie.instControllDrivers_1 := 0;
	    
	    "dbHoldRegSlave_to_MT101".Status_Sterowanie.instControllDrivers_2 := 0;
	    
	    ;
	  END_IF;
	  
	END_REGION
	
	
	REGION //Drive Motor Z6 ustaw na  Automat/Manual/Otwarta/Zamknięta
	  IF %DB58.DBX14.5 OR %DB58.DBX16.1 THEN
	    // przełączniki bistabilny każdy stan Hi powoduje zmianę przełącznika 
	    #set_aut_man_Z6 := TRUE;
	  ELSE
	    #set_aut_man_Z6 := FALSE
	    ;
	  END_IF;
	  
	  IF %DB10.DBX16.0 = FALSE THEN
	    // przełącznik bistabilny
	    "R_TRIG_DB_AUT_Z6"(CLK := #set_aut_man_Z6,
	                       Q => #setTrig_Z6);
	    ;
	  END_IF;
	  // przełącz na automat
	  IF #setTrig_Z6 = TRUE AND %DB58.DBX14.5 = TRUE THEN
	    %DB10.DBX16.7 := TRUE;
	    ;
	  END_IF;
	  // przełącz na manual
	  IF #setTrig_Z6 = TRUE AND %DB58.DBX16.1 = TRUE THEN
	    %DB10.DBX16.7 := FALSE;
	    ;
	  END_IF;
	  
	  IF (%DB10.DBX17.7 = TRUE AND %DB58.DBX14.5) OR (%DB10.DBX17.7 = FALSE AND %DB58.DBX16.1) THEN
	    // Wyczyść całą zmienną
	    "dbHoldRegSlave_to_MT101".Status_Sterowanie.instConrol_ManAut_1 := 0;
	    "dbHold_Sending".data.stat.control.control_2.set_res_bity_tryb_napędów_1 := 0;
	    "dbHoldRegSlave_to_MT101".Status_Sterowanie.instConrol_ManAut_2 := 0;
	    "dbHold_Sending".data.stat.control.control_2.set_res_bity_tryb_napędów_2 := 0;
	    %DB58.DBX14.5 := FALSE;
	    %DB58.DBX16.1 := FALSE
	    ;
	  END_IF;
	  
	  
	  // sterowanie OTWIERANIE - ZAMYKANIE
	  // Otwórz/
	  // przekazanie bitu roskazu z bloku modbus rtu do bloku statusu napędu
	  %DB10.DBX16.4 := %DB58.DBX10.5; //ustawienie bitu otwieranie
	  IF %DB58.DBX10.5 AND %DB10.DBX17.1 THEN
	    //jeśli ustawiony bit otwierania z modbus i potwierdzone otwarcie 
	    %DB58.DBX10.5 := FALSE; // kasuj bit roskazu
	    "dbHoldRegSlave_to_MT101".Status_Sterowanie.instControllDrivers_1 := 0;
	    
	    "dbHoldRegSlave_to_MT101".Status_Sterowanie.instControllDrivers_2 := 0;
	    
	    
	    ;
	  END_IF;
	  //Zamknij
	  //przekazanie bitu roskazu z bloku modbus rtu do bloku statusu napędu
	  %DB10.DBX16.5 := %DB58.DBX12.1; //ustawienie bitu zamykanie
	  IF %DB58.DBX12.1 AND %DB10.DBX17.3 = FALSE THEN
	    //jeśli ustawiony bit zamykanie z modbus i potwierdzone zamknięcie 
	    %DB58.DBX12.1 := FALSE; // kasuj bit roskazu
	    "dbHoldRegSlave_to_MT101".Status_Sterowanie.instControllDrivers_1 := 0;
	    
	    "dbHoldRegSlave_to_MT101".Status_Sterowanie.instControllDrivers_2 := 0;
	    
	    ;
	  END_IF;
	  
	END_REGION
	
	REGION //Drive Motor Z7 ustaw na  Automat/Manual/Otwarta/Zamknięta
	  IF %DB58.DBX14.6 OR %DB58.DBX16.2 THEN
	    // przełączniki bistabilny każdy stan Hi powoduje zmianę przełącznika 
	    #set_aut_man_Z7 := TRUE;
	  ELSE
	    #set_aut_man_Z7 := FALSE
	    ;
	  END_IF;
	  
	  IF %DB10.DBX18.0 = FALSE THEN
	    // przełącznik bistabilny
	    "R_TRIG_DB_AUT_Z7"(CLK := #set_aut_man_Z7,
	                       Q => #setTrig_Z7);
	    ;
	  END_IF;
	  // przełącz na automat
	  IF #setTrig_Z7 = TRUE AND %DB58.DBX14.6 = TRUE THEN
	    %DB10.DBX18.7 := TRUE;
	    ;
	  END_IF;
	  // przełącz na manual
	  IF #setTrig_Z7 = TRUE AND %DB58.DBX16.2 = TRUE THEN
	    %DB10.DBX18.7 := FALSE;
	    ;
	  END_IF;
	  
	  IF (%DB10.DBX19.7 = TRUE AND %DB58.DBX14.6) OR (%DB10.DBX19.7 = TRUE AND %DB58.DBX16.2) THEN
	    // Wyczyść całą zmienną
	    "dbHoldRegSlave_to_MT101".Status_Sterowanie.instConrol_ManAut_1 := 0;
	    "dbHold_Sending".data.stat.control.control_2.set_res_bity_tryb_napędów_1 := 0;
	    "dbHoldRegSlave_to_MT101".Status_Sterowanie.instConrol_ManAut_2 := 0;
	    "dbHold_Sending".data.stat.control.control_2.set_res_bity_tryb_napędów_2 := 0;
	    %DB58.DBX14.6 := FALSE;
	    %DB58.DBX16.2 := FALSE
	    ;
	  END_IF;
	  
	  // sterowanie OTWIERANIE - ZAMYKANIE
	  // Otwórz/
	  // przekazanie bitu roskazu z bloku modbus rtu do bloku statusu napędu
	  %DB10.DBX18.4 := %DB58.DBX10.6; //ustawienie bitu otwieranie
	  IF %DB58.DBX10.6 AND %DB10.DBX19.1 THEN
	    //jeśli ustawiony bit otwierania z modbus i potwierdzone otwarcie 
	    %DB58.DBX10.6 := FALSE; // kasuj bit roskazu
	    "dbHoldRegSlave_to_MT101".Status_Sterowanie.instControllDrivers_1 := 0;
	    
	    "dbHoldRegSlave_to_MT101".Status_Sterowanie.instControllDrivers_2 := 0;
	    
	    
	    ;
	  END_IF;
	  //Zamknij
	  //przekazanie bitu roskazu z bloku modbus rtu do bloku statusu napędu
	  %DB10.DBX18.5 := %DB58.DBX12.2; //ustawienie bitu zamykanie
	  IF %DB58.DBX12.2 AND %DB10.DBX19.3 = FALSE THEN
	    //jeśli ustawiony bit zamykanie z modbus i potwierdzone zamknięcie 
	    %DB58.DBX12.2 := FALSE; // kasuj bit roskazu
	    "dbHoldRegSlave_to_MT101".Status_Sterowanie.instControllDrivers_1 := 0;
	    
	    "dbHoldRegSlave_to_MT101".Status_Sterowanie.instControllDrivers_2 := 0;
	    
	    ;
	  END_IF;
	  
	END_REGION
	
	
	
	
	REGION //Drive Motor Z8 ustaw na  Automat/Manual/Otwarta/Zamknięta
	  IF %DB58.DBX14.7 OR %DB58.DBX16.3 THEN
	  // przełączniki bistabilny każdy stan Hi powoduje zmianę przełącznika 
	    #set_aut_man_Z8 := TRUE;
	  ELSE
	    #set_aut_man_Z8:= FALSE
	  ;
	END_IF;
	
	IF %DB10.DBX20.0 = FALSE THEN
	  // przełącznik bistabilny
	  "R_TRIG_DB_AUT_Z8"(CLK := #set_aut_man_Z8,
	                     Q => #setTrig_Z8);
	  ;
	END_IF;
	// przełącz na automat
	IF #setTrig_Z8 = TRUE AND %DB58.DBX14.7 = TRUE THEN
	  %DB10.DBX20.7 := TRUE;
	  ;
	END_IF;
	// przełącz na manual 
	IF #setTrig_Z8 = TRUE AND %DB58.DBX16.3 = TRUE THEN
	  %DB10.DBX20.7 := FALSE;
	  ;
	END_IF;
	
	IF (%DB10.DBX21.7 = TRUE AND %DB58.DBX14.7) OR (%DB10.DBX21.7 = FALSE AND %DB58.DBX16.3) THEN
	  // Wyczyść całą zmienną
	  "dbHoldRegSlave_to_MT101".Status_Sterowanie.instConrol_ManAut_1 := 0;
	  "dbHold_Sending".data.stat.control.control_2.set_res_bity_tryb_napędów_1 := 0;
	  "dbHoldRegSlave_to_MT101".Status_Sterowanie.instConrol_ManAut_2 := 0;
	  "dbHold_Sending".data.stat.control.control_2.set_res_bity_tryb_napędów_2 := 0;
	  %DB58.DBX14.7 := FALSE;
	  %DB58.DBX16.3 := FALSE
	  ;
	END_IF;
	
	// sterowanie OTWIERANIE - ZAMYKANIE
	// Otwórz/
	// przekazanie bitu roskazu z bloku modbus rtu do bloku statusu napędu
	%DB10.DBX20.4 := %DB58.DBX10.7; //ustawienie bitu otwieranie
	IF %DB58.DBX10.7 AND %DB10.DBX21.1 THEN
	  //jeśli ustawiony bit otwierania z modbus i potwierdzone otwarcie 
	  %DB58.DBX10.7 := FALSE; // kasuj bit roskazu
	  "dbHoldRegSlave_to_MT101".Status_Sterowanie.instControllDrivers_1 := 0;
	  
	  "dbHoldRegSlave_to_MT101".Status_Sterowanie.instControllDrivers_2 := 0;
	  
	  
	  ;
	END_IF;
	//Zamknij
	//przekazanie bitu roskazu z bloku modbus rtu do bloku statusu napędu
	%DB10.DBX20.5 := %DB58.DBX12.3; //ustawienie bitu zamykanie
	IF %DB58.DBX12.3 AND %DB10.DBX21.3 = FALSE THEN
	  //jeśli ustawiony bit zamykanie z modbus i potwierdzone zamknięcie 
	  %DB58.DBX12.3 := FALSE; // kasuj bit roskazu
	  "dbHoldRegSlave_to_MT101".Status_Sterowanie.instControllDrivers_1 := 0;
	  
	  "dbHoldRegSlave_to_MT101".Status_Sterowanie.instControllDrivers_2 := 0;
	  
	  ;
	END_IF;
	  
	END_REGION
	
	
	REGION //Drive Motor Z9 ustaw na  Automat/Manual/Otwarta/Zamknięta
	  IF %DB58.DBX17.0  OR %DB58.DBX16.4THEN
	    //przełączniki bistabilny każdy stan Hi powoduje zmianę przełącznika 
	    #set_aut_man_Z9 := TRUE;
	  ELSE
	    #set_aut_man_Z9:= FALSE
	    ;
	  END_IF;
	  IF %DB10.DBX22.0 = FALSE THEN
	    // przełaącznik bistabilny
	    "R_TRIG_DB_AUT_Z9"(CLK := #set_aut_man_Z9,
	                       Q => #setTrig_Z9);
	    ;
	  END_IF;
	  // przełąćż na automat
	  IF #setTrig_Z9 = TRUE AND %DB58.DBX17.0 = TRUE THEN
	    %DB10.DBX22.7 := TRUE;
	    ;
	  END_IF;
	  // przełąćż na manual
	  IF #setTrig_Z9 = TRUE AND %DB58.DBX16.4 = TRUE THEN
	    %DB10.DBX22.7 := FALSE;
	    ;
	  END_IF;
	  
	  IF (%DB10.DBX23.7 = TRUE AND %DB58.DBX17.0) OR (%DB10.DBX23.7 = TRUE AND %DB58.DBX16.4) THEN
	    // Wyczyść całą zmienną
	    "dbHoldRegSlave_to_MT101".Status_Sterowanie.instConrol_ManAut_2 := 0;
	    "dbHold_Sending".data.stat.control.control_2.set_res_bity_tryb_napędów_2 := 0;
	    %DB58.DBX17.0 := FALSE;
	    %DB58.DBX16.4 := FALSE
	    ;
	  END_IF;
	  
	  // sterowanie OTWIERANIE - ZAMYKANIE
	  // Otwórz/
	  // przekazanie bitu roskazu z bloku modbus rtu do bloku statusu napędu
	  %DB10.DBX22.4 := %DB58.DBX13.0; //ustawienie bitu otwieranie
	  IF %DB58.DBX13.0 AND %DB10.DBX23.1 THEN
	    //jeśli ustawiony bit otwierania z modbus i potwierdzone otwarcie 
	    %DB58.DBX13.0 := FALSE; // kasuj bit roskazu
	    "dbHoldRegSlave_to_MT101".Status_Sterowanie.instControllDrivers_1 := 0;
	    
	    "dbHoldRegSlave_to_MT101".Status_Sterowanie.instControllDrivers_2 := 0;
	    
	    
	    ;
	  END_IF;
	  //Zamknij
	  //przekazanie bitu roskazu z bloku modbus rtu do bloku statusu napędu
	  %DB10.DBX22.5 := %DB58.DBX12.4; //ustawienie bitu zamykanie
	  IF %DB58.DBX12.4 AND %DB10.DBX23.3 = FALSE THEN
	    //jeśli ustawiony bit zamykanie z modbus i potwierdzone zamknięcie 
	    %DB58.DBX12.4 := FALSE; // kasuj bit roskazu
	    "dbHoldRegSlave_to_MT101".Status_Sterowanie.instControllDrivers_1 := 0;
	    
	    "dbHoldRegSlave_to_MT101".Status_Sterowanie.instControllDrivers_2 := 0;
	    
	    ;
	  END_IF;
	  
	END_REGION
	
	
	REGION //Drive Motor Z10 ustaw na  Automat/Manual/Otwarta/Zamknięta
	  IF %DB58.DBX17.1 OR %DB58.DBX16.5 THEN
	    //przełączniki bistabilny każdy stan Hi powoduje zmianę przełącznika 
	    #set_aut_man_Z10 := TRUE;
	  ELSE
	    #set_aut_man_Z10:= FALSE
	  ;
	END_IF;
	IF %DB10.DBX24.0 = FALSE THEN
	  // przełącznik bistabilny
	  "R_TRIG_DB_AUT_Z10"(CLK := #set_aut_man_Z10,
	                      Q => #setTrig_Z10);
	  ;
	END_IF;
	// przełącz na automat
	IF #setTrig_Z10 = TRUE AND %DB58.DBX17.1 = TRUE THEN
	  %DB10.DBX24.7 := TRUE;
	  ;
	END_IF;
	// przełącz na manual
	IF #setTrig_Z10 = TRUE AND %DB58.DBX16.5 = TRUE THEN
	  %DB10.DBX24.7 := FALSE;
	  ;
	END_IF;
	
	IF (%DB10.DBX25.7 = TRUE AND %DB58.DBX17.1) OR (%DB10.DBX25.7 = FALSE AND %DB58.DBX16.5) THEN
	  // Wyczyść całą zmienną
	  "dbHoldRegSlave_to_MT101".Status_Sterowanie.instConrol_ManAut_2 := 0;
	  "dbHold_Sending".data.stat.control.control_2.set_res_bity_tryb_napędów_2 := 0;
	  %DB58.DBX17.0 := FALSE;
	  %DB58.DBX16.5 := FALSE
	  ;
	END_IF;
	
	// sterowanie OTWIERANIE - ZAMYKANIE
	// Otwórz/
	// przekazanie bitu roskazu z bloku modbus rtu do bloku statusu napędu
	%DB10.DBX24.4 := %DB58.DBX13.1; //ustawienie bitu otwieranie
	IF %DB58.DBX13.1 AND %DB10.DBX25.1 THEN
	  //jeśli ustawiony bit otwierania z modbus i potwierdzone otwarcie 
	  %DB58.DBX13.1 := FALSE; // kasuj bit roskazu
	  "dbHoldRegSlave_to_MT101".Status_Sterowanie.instControllDrivers_1 := 0;
	  
	  "dbHoldRegSlave_to_MT101".Status_Sterowanie.instControllDrivers_2 := 0;
	  
	  
	  ;
	END_IF;
	//Zamknij
	//przekazanie bitu roskazu z bloku modbus rtu do bloku statusu napędu
	%DB10.DBX24.5 := %DB58.DBX12.5; //ustawienie bitu zamykanie
	IF %DB58.DBX12.5 AND %DB10.DBX25.3 = FALSE THEN
	  //jeśli ustawiony bit zamykanie z modbus i potwierdzone zamknięcie 
	  %DB58.DBX12.5 := FALSE; // kasuj bit roskazu
	  "dbHoldRegSlave_to_MT101".Status_Sterowanie.instControllDrivers_1 := 0;
	  
	  "dbHoldRegSlave_to_MT101".Status_Sterowanie.instControllDrivers_2 := 0;
	  
	  ;
	END_IF;
	  
	END_REGION
	
	
	
	
	
	
	
	
	
	
	
	
	
END_FUNCTION_BLOCK

FUNCTION "Błąd Modbus TCP" : Void
TITLE = Obsługa błędu
{ S7_Optimized_Access := 'TRUE' }
AUTHOR : rtecmer
VERSION : 0.1
//Funkcja ubsługuje zainicjowany błąd komunikacji Modbus TCP
   VAR_INPUT 
      bit_loop : Bool;   // znacznik ostatniego bloku pętli
   END_VAR

   VAR_IN_OUT 
      "bit_reset-modbus_tcp" : Bool;   // bit restartu modbus tcp
   END_VAR

   VAR_TEMP 
      reset : Bool;
      reset_1 : Bool;
   END_VAR


BEGIN
	(*
	//=============================================================================
	//(JZWiK S.A Radosław Tecmer)
	//(c)Copyright (2022) All Rights Reserved
	//-----------------------------------------------------------------------------
	//Testowane z:   (system docelowy z  FW 4.4)
	//Pakiet inżynierski:   TIA Portal (V16 Update 5)
	//Ograniczenia:  ( - )
	//Wymagania:  (minimalne S7-1200 CPU 1215C FW 4.2 .)
	//Funkcjonalnośc: (Funkcja ubsługuje zainicjowany błąd komunikacji Modbus TCP )
	//-----------------------------------------------------------------------------
	//Zmainy wprowadzone:
	//Wersja  Data       Osoba wprowadzająca zmiany - ekspert
	//01.00.00 09.03.2022 (Tecmer Radosław - twórca) Pieresza wersja 01.00.00
	//=============================================================================
	*)
	
	
	
	
	REGION Kontrola staru Modbus TCP
	  // histereza na start 
	  IF ("DB31_HMI_AreaPointer".cpuSatus = FALSE) AND ("DB31_HMI_AreaPointer".getPLCMode = 2) THEN
	    // uruchom timer startu tcp
	    "memRisingTriger_tmerDisconected" := TRUE;
	    ;
	  END_IF;
	  
	  
	END_REGION
	
	
	// Jeśli wystąpi błąd to reset
	IF "MB_TCP_CLIENT".MB_Client_Receiving.Input.InOut.error
	  OR "MB_TCP_CLIENT".MB_Client_Receiving_Time.Input.InOut.error
	  OR "MB_TCP_CLIENT".MB_Client_Receiving_Time.Input.InOut.error
	  OR "MB_TCP_CLIENT".MB_Client_Sending.Input.InOut.error
	  OR "MB_TCP_CLIENT".MB_Client_Sending_1.Input.InOut.error
	  OR "MB_TCP_CLIENT".MB_Client_Sending_3.Input.InOut.error
	  
	THEN
	  // Reset komunikacji
	  "MB_TCP_CLIENT".MB_Client_Sending.Input.disconnect := TRUE;
	  "MB_TCP_CLIENT".MB_Client_Receiving_Time.Input.disconnect:= TRUE;
	  "MB_TCP_CLIENT".MB_Client_Sending_1.Input.disconnect := TRUE;
	  "MB_TCP_CLIENT".MB_Client_Sending_3.Input.disconnect := TRUE;
	  "MB_TCP_CLIENT".MB_Client_Receiving.Input.disconnect := FALSE;
	  "done_modbusTCP_przetw_1" := TRUE;
	  "done_modbusTCP_przetw_2" := FALSE;
	  "done_modbusTCP_przetw_3" := FALSE;
	  "done_modbusTCP_przetw_4" := FALSE;
	  "done_modbusTCP_przetw_5" := FALSE;
	  "MB_TCP_CLIENT".MB_Client_Receiving.tagsStep.step := 1;
	  "MB_TCP_CLIENT".MB_Client_Sending_1.tagsStep.step := 0;
	  "MB_TCP_CLIENT".MB_Client_Receiving_Time.tagsStep.step := 0;
	  "MB_TCP_CLIENT".MB_Client_Sending.tagsStep.step := 0;
	  "MB_TCP_CLIENT".MB_Client_Sending_3.tagsStep.step := 0;
	  "MB_TCP_CLIENT".MB_Client_Receiving.Input.InOut.error := FALSE;
	  "MB_TCP_CLIENT".MB_Client_Receiving_Time.Input.InOut.error := FALSE;
	  "MB_TCP_CLIENT".MB_Client_Sending.Input.InOut.error := FALSE;
	  "MB_TCP_CLIENT".MB_Client_Sending_2.Input.InOut.error := FALSE;
	  "MB_TCP_CLIENT".MB_Client_Sending_3.Input.InOut.error := FALSE;
	  "MB_TCP_CLIENT".MB_Client_Sending_4.Input.InOut.error := FALSE;
	  "MB_TCP_CLIENT".MB_Client_Receiving.Input.InOut.ERROR_STATUS := 0;
	  "MB_TCP_CLIENT".MB_Client_Receiving_Time.Input.InOut.ERROR_STATUS := 0;
	  "MB_TCP_CLIENT".MB_Client_Sending.Input.InOut.ERROR_STATUS := 0;
	  "MB_TCP_CLIENT".MB_Client_Sending_2.Input.InOut.ERROR_STATUS := 0;
	  "MB_TCP_CLIENT".MB_Client_Sending_3.Input.InOut.ERROR_STATUS := 0;
	  "MB_TCP_CLIENT".MB_Client_Sending_4.Input.InOut.ERROR_STATUS := 0;
	  "memRisingTriger_Data_1" := FALSE;
	  "memRisingTriger_Data_2" := FALSE;
	  "memRisingTriger_Data_3" := FALSE;
	  "memRisingTriger_Data_4" := FALSE;
	  "memRisingTriger_Data_5" := FALSE;
	  "memRisingTriger_Data_6" := FALSE;
	  "memRisingTriger_Data_7" := FALSE;
	  "memRisingTriger_Data_8" := FALSE;
	  "memRisingTriger_Data_9" := FALSE;
	  "memRisingTriger_Data_10" := FALSE;
	  "memRisingTriger_Data_11" := FALSE;
	  "memRisingTriger_Data_12" := FALSE;
	  "memRisingTriger_Data_13" := FALSE;
	  "memRisingTriger_Data_14" := FALSE;
	  "memRisingTriger_Data_15" := FALSE;
	  "memRisingTriger_Data_16" := FALSE;
	  "memTrig_Client_Receiving_1" := FALSE;
	  "memTrig_Client_Receiving_2" := FALSE;
	  "memTrig_Client_Receiving_3" := FALSE;
	  "memTrig_Client_Receiving_4" := FALSE;
	  "memTrig_Client_Receiving_5" := FALSE;
	  "memTrig_Client_Receiving_7" := FALSE;
	  "memTrig_Client_Receiving_8" := FALSE;
	  "memTrig_Client_Receiving_9" := FALSE;
	  "memTrig_Client_Receiving_10" := FALSE;
	  "memTrig_Client_Receiving_11" := FALSE;
	  "memTrig_Client_Receiving_12" := FALSE;
	  "memTrig_Client_Receiving_13" := FALSE;
	  "memTrig_Client_Receiving_14" := FALSE;
	  "memTrig_Client_Receiving_15" := FALSE;
	  "memTrig_Client_Receiving_16" := FALSE;
	  
	END_IF;
	
	// Jesli pętla MOdbus TCP błąd obiegu
	IF "done_modbusTCP_przetw_1" = FALSE
	  AND "done_modbusTCP_przetw_2" = FALSE
	  AND "done_modbusTCP_przetw_3" = FALSE
	  AND "done_modbusTCP_przetw_4" = FALSE
	  AND "done_modbusTCP_przetw_5" = FALSE
	THEN
	  "done_modbusTCP_przetw_1":= TRUE
	  
	  ;
	END_IF;
	
	//Kasowanie błedu jesli brak bitu error
	
	// blok pobierania sterowania
	IF ("MB_TCP_CLIENT".MB_Client_Receiving.Input.InOut.ERROR_STATUS <> 0)
	  AND "MB_TCP_CLIENT".MB_Client_Receiving.Input.InOut.error = FALSE
	THEN
	  //kasuj błąd
	  "MB_TCP_CLIENT".MB_Client_Receiving.Input.InOut.ERROR_STATUS := 0;
	  "memRisingTriger_Data_1" := FALSE;
	  "memRisingTriger_Data_2" := FALSE;
	  "memRisingTriger_Data_3" := FALSE;
	  "memRisingTriger_Data_4" := FALSE;
	  "memRisingTriger_Data_5" := FALSE;
	  "memRisingTriger_Data_6" := FALSE;
	  "memRisingTriger_Data_7" := FALSE;
	  "memRisingTriger_Data_8" := FALSE;
	  "memRisingTriger_Data_9" := FALSE;
	  "memRisingTriger_Data_10" := FALSE;
	  "memRisingTriger_Data_11" := FALSE;
	  "memRisingTriger_Data_12" := FALSE;
	  "memRisingTriger_Data_13" := FALSE;
	  "memRisingTriger_Data_14" := FALSE;
	  "memRisingTriger_Data_15" := FALSE;
	  "memRisingTriger_Data_16" := FALSE;
	  "memTrig_Client_Receiving_1" := FALSE;
	  "memTrig_Client_Receiving_2" := FALSE;
	  "memTrig_Client_Receiving_3" := FALSE;
	  "memTrig_Client_Receiving_4" := FALSE;
	  "memTrig_Client_Receiving_5" := FALSE;
	  "memTrig_Client_Receiving_7" := FALSE;
	  "memTrig_Client_Receiving_8" := FALSE;
	  "memTrig_Client_Receiving_9" := FALSE;
	  "memTrig_Client_Receiving_10" := FALSE;
	  "memTrig_Client_Receiving_11" := FALSE;
	  "memTrig_Client_Receiving_12" := FALSE;
	  "memTrig_Client_Receiving_13" := FALSE;
	  "memTrig_Client_Receiving_14" := FALSE;
	  "memTrig_Client_Receiving_15" := FALSE;
	  "memTrig_Client_Receiving_16" := FALSE;
	  ;
	END_IF;
	
	// blok pobierania DTL
	IF ("MB_TCP_CLIENT".MB_Client_Receiving_Time.Input.InOut.ERROR_STATUS <> 0)
	  AND "MB_TCP_CLIENT".MB_Client_Receiving_Time.Input.InOut.error = FALSE
	THEN
	  //kasuj błąd
	  "MB_TCP_CLIENT".MB_Client_Receiving_Time.Input.InOut.ERROR_STATUS := 0;
	  "memRisingTriger_Data_1" := FALSE;
	  "memRisingTriger_Data_2" := FALSE;
	  "memRisingTriger_Data_3" := FALSE;
	  "memRisingTriger_Data_4" := FALSE;
	  "memRisingTriger_Data_5" := FALSE;
	  "memRisingTriger_Data_6" := FALSE;
	  "memRisingTriger_Data_7" := FALSE;
	  "memRisingTriger_Data_8" := FALSE;
	  "memRisingTriger_Data_9" := FALSE;
	  "memRisingTriger_Data_10" := FALSE;
	  "memRisingTriger_Data_11" := FALSE;
	  "memRisingTriger_Data_12" := FALSE;
	  "memRisingTriger_Data_13" := FALSE;
	  "memRisingTriger_Data_14" := FALSE;
	  "memRisingTriger_Data_15" := FALSE;
	  "memRisingTriger_Data_16" := FALSE;
	  "memTrig_Client_Receiving_1" := FALSE;
	  "memTrig_Client_Receiving_2" := FALSE;
	  "memTrig_Client_Receiving_3" := FALSE;
	  "memTrig_Client_Receiving_4" := FALSE;
	  "memTrig_Client_Receiving_5" := FALSE;
	  "memTrig_Client_Receiving_7" := FALSE;
	  "memTrig_Client_Receiving_8" := FALSE;
	  "memTrig_Client_Receiving_9" := FALSE;
	  "memTrig_Client_Receiving_10" := FALSE;
	  "memTrig_Client_Receiving_11" := FALSE;
	  "memTrig_Client_Receiving_12" := FALSE;
	  "memTrig_Client_Receiving_13" := FALSE;
	  "memTrig_Client_Receiving_14" := FALSE;
	  "memTrig_Client_Receiving_15" := FALSE;
	  "memTrig_Client_Receiving_16" := FALSE;
	  ;
	END_IF;
	
	// blok wysyłania analogów
	IF ("MB_TCP_CLIENT".MB_Client_Sending.Input.InOut.ERROR_STATUS <> 0)
	  AND "MB_TCP_CLIENT".MB_Client_Sending.Input.InOut.error = FALSE
	THEN
	  //kasuj błąd
	  "MB_TCP_CLIENT".MB_Client_Sending.Input.InOut.ERROR_STATUS := 0;
	  "memRisingTriger_Data_1" := FALSE;
	  "memRisingTriger_Data_2" := FALSE;
	  "memRisingTriger_Data_3" := FALSE;
	  "memRisingTriger_Data_4" := FALSE;
	  "memRisingTriger_Data_5" := FALSE;
	  "memRisingTriger_Data_6" := FALSE;
	  "memRisingTriger_Data_7" := FALSE;
	  "memRisingTriger_Data_8" := FALSE;
	  "memRisingTriger_Data_9" := FALSE;
	  "memRisingTriger_Data_10" := FALSE;
	  "memRisingTriger_Data_11" := FALSE;
	  "memRisingTriger_Data_12" := FALSE;
	  "memRisingTriger_Data_13" := FALSE;
	  "memRisingTriger_Data_14" := FALSE;
	  "memRisingTriger_Data_15" := FALSE;
	  "memRisingTriger_Data_16" := FALSE;
	  "memTrig_Client_Receiving_1" := FALSE;
	  "memTrig_Client_Receiving_2" := FALSE;
	  "memTrig_Client_Receiving_3" := FALSE;
	  "memTrig_Client_Receiving_4" := FALSE;
	  "memTrig_Client_Receiving_5" := FALSE;
	  "memTrig_Client_Receiving_7" := FALSE;
	  "memTrig_Client_Receiving_8" := FALSE;
	  "memTrig_Client_Receiving_9" := FALSE;
	  "memTrig_Client_Receiving_10" := FALSE;
	  "memTrig_Client_Receiving_11" := FALSE;
	  "memTrig_Client_Receiving_12" := FALSE;
	  "memTrig_Client_Receiving_13" := FALSE;
	  "memTrig_Client_Receiving_14" := FALSE;
	  "memTrig_Client_Receiving_15" := FALSE;
	  "memTrig_Client_Receiving_16" := FALSE;
	  ;
	END_IF;
	
	// blok wysyłąnia statusów
	IF ("MB_TCP_CLIENT".MB_Client_Sending_1.Input.InOut.ERROR_STATUS <> 0)
	  AND "MB_TCP_CLIENT".MB_Client_Sending_1.Input.InOut.error = FALSE
	THEN
	  //kasuj błąd
	  "MB_TCP_CLIENT".MB_Client_Sending_1.Input.InOut.ERROR_STATUS := 0;
	  "memRisingTriger_Data_1" := FALSE;
	  "memRisingTriger_Data_2" := FALSE;
	  "memRisingTriger_Data_3" := FALSE;
	  "memRisingTriger_Data_4" := FALSE;
	  "memRisingTriger_Data_5" := FALSE;
	  "memRisingTriger_Data_6" := FALSE;
	  "memRisingTriger_Data_7" := FALSE;
	  "memRisingTriger_Data_8" := FALSE;
	  "memRisingTriger_Data_9" := FALSE;
	  "memRisingTriger_Data_10" := FALSE;
	  "memRisingTriger_Data_11" := FALSE;
	  "memRisingTriger_Data_12" := FALSE;
	  "memRisingTriger_Data_13" := FALSE;
	  "memRisingTriger_Data_14" := FALSE;
	  "memRisingTriger_Data_15" := FALSE;
	  "memRisingTriger_Data_16" := FALSE;
	  "memTrig_Client_Receiving_1" := FALSE;
	  "memTrig_Client_Receiving_2" := FALSE;
	  "memTrig_Client_Receiving_3" := FALSE;
	  "memTrig_Client_Receiving_4" := FALSE;
	  "memTrig_Client_Receiving_5" := FALSE;
	  "memTrig_Client_Receiving_7" := FALSE;
	  "memTrig_Client_Receiving_8" := FALSE;
	  "memTrig_Client_Receiving_9" := FALSE;
	  "memTrig_Client_Receiving_10" := FALSE;
	  "memTrig_Client_Receiving_11" := FALSE;
	  "memTrig_Client_Receiving_12" := FALSE;
	  "memTrig_Client_Receiving_13" := FALSE;
	  "memTrig_Client_Receiving_14" := FALSE;
	  "memTrig_Client_Receiving_15" := FALSE;
	  "memTrig_Client_Receiving_16" := FALSE;
	  ;
	END_IF;
	
	// blok wysyłania parametrów
	IF ("MB_TCP_CLIENT".MB_Client_Sending_3.Input.InOut.ERROR_STATUS <> 0)
	  AND "MB_TCP_CLIENT".MB_Client_Sending_3.Input.InOut.error = FALSE
	THEN
	  //kasuj błąd
	  "MB_TCP_CLIENT".MB_Client_Sending_3.Input.InOut.ERROR_STATUS := 0;
	  "memRisingTriger_Data_1" := FALSE;
	  "memRisingTriger_Data_2" := FALSE;
	  "memRisingTriger_Data_3" := FALSE;
	  "memRisingTriger_Data_4" := FALSE;
	  "memRisingTriger_Data_5" := FALSE;
	  "memRisingTriger_Data_6" := FALSE;
	  "memRisingTriger_Data_7" := FALSE;
	  "memRisingTriger_Data_8" := FALSE;
	  "memRisingTriger_Data_9" := FALSE;
	  "memRisingTriger_Data_10" := FALSE;
	  "memRisingTriger_Data_11" := FALSE;
	  "memRisingTriger_Data_12" := FALSE;
	  "memRisingTriger_Data_13" := FALSE;
	  "memRisingTriger_Data_14" := FALSE;
	  "memRisingTriger_Data_15" := FALSE;
	  "memRisingTriger_Data_16" := FALSE;
	  "memTrig_Client_Receiving_1" := FALSE;
	  "memTrig_Client_Receiving_2" := FALSE;
	  "memTrig_Client_Receiving_3" := FALSE;
	  "memTrig_Client_Receiving_4" := FALSE;
	  "memTrig_Client_Receiving_5" := FALSE;
	  "memTrig_Client_Receiving_7" := FALSE;
	  "memTrig_Client_Receiving_8" := FALSE;
	  "memTrig_Client_Receiving_9" := FALSE;
	  "memTrig_Client_Receiving_10" := FALSE;
	  "memTrig_Client_Receiving_11" := FALSE;
	  "memTrig_Client_Receiving_12" := FALSE;
	  "memTrig_Client_Receiving_13" := FALSE;
	  "memTrig_Client_Receiving_14" := FALSE;
	  "memTrig_Client_Receiving_15" := FALSE;
	  "memTrig_Client_Receiving_16" := FALSE;
	  ;
	END_IF;
	
	
	IF ("Clock_0.625Hz" = TRUE) AND ("memTrig_loop_error" = TRUE)   THEN
	  // Aktywuj błąd przerwanie pętli modbu tcp
	  "Dane_ComunicationControlHMI"."CoordinationPLC-PLC" := 24;
	  ;
	END_IF;
	
	
	
	
	
	
	#reset := FALSE;
	
	
END_FUNCTION

FUNCTION_BLOCK "alarm_petli-rtu_tcp"   // FB14, LAD
TITLE = kontrola obiegu pętli rtu, tcp
{ S7_Optimized_Access := 'TRUE' }
AUTHOR : rtecmer
VERSION : 0.1
// jeśli pętla się zawiesi bez sygnałizacji błędu w statusie to po ustalonym czasie 2x czas obiegu pętli nastąpi ustawienie znaczniku awaria pętli
// stored: AutoNumber true, IsIECCheckEnabled false, IsRetainMemResEnabled false, MemoryReserve 100, SetENOAutomatically false, UDAEnableTagReadback false
BEGIN

REGION Network 1: błąd petli Modbus TCP brak obiegu pętli
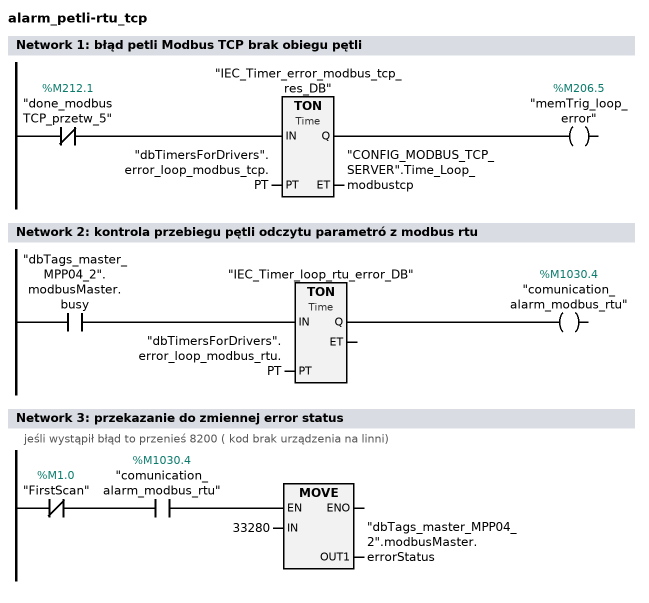
   RUNG wire#powerrail
      I_Contact( "done_modbusTCP_przetw_5" )
      { S7_Templates := "time_type := Time" } "IEC_Timer_error_modbus_tcp_res_DB".TON(pt := "dbTimersForDrivers".error_loop_modbus_tcp.PT, et => "CONFIG_MODBUS_TCP_SERVER".Time_Loop_modbustcp)
      Coil( "memTrig_loop_error" )
   END_RUNG
   // the same network as SCL:
   "IEC_Timer_error_modbus_tcp_res_DB".TON(IN := NOT "done_modbusTCP_przetw_5",
                           PT := "dbTimersForDrivers".error_loop_modbus_tcp.PT,
                           ET => "CONFIG_MODBUS_TCP_SERVER".Time_Loop_modbustcp);
   "memTrig_loop_error" := "IEC_Timer_error_modbus_tcp_res_DB".Q;
END_REGION

